LIN {X 0,Y 171.569,Z 534.537,A -85,B 0,C 180,E1 -24803.925,E2 -24803.925} C_VEL
LIN {X 0,Y 171.044,Z 531.437,A -85,B 0,C 180,E1 -24804.883,E2 -24804.883} C_VEL
LIN {X 0,Y 169.506,Z 526.594,A -85,B 0,C 180,E1 -24806.675,E2 -24806.675} C_VEL
LIN {X 0,Y 166.044,Z 528.715,A -85,B 0,C 180,E1 -24808.057,E2 -24808.057} C_VEL
LIN {X 0,Y 163.92,Z 529.698,A -85,B 0,C 180,E1 -24809.036,E2 -24809.036} C_VEL
LIN {X 0,Y 158.88,Z 534.272,A -85,B 0,C 180,E1 -24810.884,E2 -24810.884} C_VEL
LIN {X 0,Y 156.535,Z 535.959,A -85,B 0,C 180,E1 -24811.94,E2 -24811.94} C_VEL
LIN {X 0,Y 150.862,Z 538.736,A -85,B 0,C 180,E1 -24815.211,E2 -24815.211} C_VEL
LIN {X 0,Y 146.783,Z 541.804,A -85,B 0,C 180,E1 -24817.477,E2 -24817.477} C_VEL
LIN {X 0,Y 140.545,Z 545.035,A -85,B 0,C 180,E1 -24822.54,E2 -24822.54} C_VEL
LIN {X 0,Y 139.213,Z 546.109,A -85,B 0,C 180,E1 -24823.576,E2 -24823.576} C_VEL
LIN {X 0,Y 137.537,Z 547.231,A -85,B 0,C 180,E1 -24825.197,E2 -24825.197} C_VEL
LIN {X 0,Y 135.805,Z 547.355,A -85,B 0,C 180,E1 -24828.261,E2 -24828.261} C_VEL
LIN {X 0,Y 135.037,Z 555.759,A -85,B 0,C 180,E1 -24834.025,E2 -24834.025} C_VEL
LIN {X 0,Y 134.715,Z 562.924,A -85,B 0,C 180,E1 -24840,E2 -24840} C_VEL
LIN {X 0,Y 136.036,Z 570.119,A -85,B 0,C 180,E1 -24847.421,E2 -24847.421} C_VEL
LIN {X 0,Y 138.515,Z 574.658,A -85,B 0,C 180,E1 -24853.198,E2 -24853.198} C_VEL
LIN {X 0,Y 143.17,Z 578.949,A -85,B 0,C 180,E1 -24860.097,E2 -24860.097} C_VEL
LIN {X 0,Y 148.115,Z 581.35,A -85,B 0,C 180,E1 -24865.28,E2 -24865.28} C_VEL
LIN {X 0,Y 154.373,Z 582.922,A -85,B 0,C 180,E1 -24870.052,E2 -24870.052} C_VEL
LIN {X 0,Y 161.797,Z 583.682,A -85,B 0,C 180,E1 -24874.38,E2 -24874.38} C_VEL
LIN {X 0,Y 170.253,Z 583.595,A -85,B 0,C 180,E1 -24878.257,E2 -24878.257} C_VEL
LIN {X 0,Y 179.651,Z 582.767,A -85,B 0,C 180,E1 -24881.686,E2 -24881.686} C_VEL
LIN {X 0,Y 179.681,Z 582.884,A -85,B 0,C 180,E1 -24881.999,E2 -24881.999} C_VEL
LIN {X 0,Y 165.118,Z 588.068,A -85,B 0,C 180,E1 -24887.077,E2 -24887.077} C_VEL
LIN {X 0,Y 158.02,Z 590.446,A -85,B 0,C 180,E1 -24890.361,E2 -24890.361} C_VEL
LIN {X 0,Y 152.368,Z 599.787,A -85,B 0,C 180,E1 -24893.978,E2 -24893.978} C_VEL
LIN {X 0,Y 146.919,Z 608.149,A -85,B 0,C 180,E1 -24898.251,E2 -24898.251} C_VEL
LIN {X 0,Y 142.926,Z 614.092,A -85,B 0,C 180,E1 -24902.264,E2 -24902.264} C_VEL
LIN {X 0,Y 139.782,Z 618.749,A -85,B 0,C 180,E1 -24906.283,E2 -24906.283} C_VEL
LIN {X 0,Y 136.398,Z 623.68,A -85,B 0,C 180,E1 -24911.992,E2 -24911.992} C_VEL
LIN {X 0,Y 134.421,Z 627.109,A -85,B 0,C 180,E1 -24917.928,E2 -24917.928} C_VEL
LIN {X 0,Y 133.541,Z 629.139,A -85,B 0,C 180,E1 -24923.958,E2 -24923.958} C_VEL
LIN {X 0,Y 133.456,Z 629.808,A -85,B 0,C 180,E1 -24930,E2 -24930} C_VEL
LIN {X 0,Y 133.541,Z 629.118,A -85,B 0,C 180,E1 -24936.042,E2 -24936.042} C_VEL
LIN {X 0,Y 134.414,Z 627.073,A -85,B 0,C 180,E1 -24942.072,E2 -24942.072} C_VEL
LIN {X 0,Y 136.386,Z 623.622,A -85,B 0,C 180,E1 -24948.01,E2 -24948.01} C_VEL
LIN {X 0,Y 139.73,Z 618.666,A -85,B 0,C 180,E1 -24953.727,E2 -24953.727} C_VEL
LIN {X 0,Y 144.19,Z 612.057,A -85,B 0,C 180,E1 -24959.171,E2 -24959.171} C_VEL
LIN {X 0,Y 149.133,Z 604.663,A -85,B 0,C 180,E1 -24963.623,E2 -24963.623} C_VEL
LIN {X 0,Y 153.97,Z 596.923,A -85,B 0,C 180,E1 -24967.214,E2 -24967.214} C_VEL
LIN {X 0,Y 155.689,Z 594.039,A -85,B 0,C 180,E1 -24968.331,E2 -24968.331} C_VEL
LIN {X 0,Y 157.521,Z 590.227,A -85,B 0,C 180,E1 -24969.845,E2 -24969.845} C_VEL
LIN {X 0,Y 159.212,Z 583.792,A -85,B 0,C 180,E1 -24972.497,E2 -24972.497} C_VEL
LIN {X 0,Y 160.162,Z 578.388,A -85,B 0,C 180,E1 -24974.587,E2 -24974.587} C_VEL
LIN {X 0,Y 161.493,Z 572.56,A -85,B 0,C 180,E1 -24976.473,E2 -24976.473} C_VEL
LIN {X 0,Y 164.734,Z 560.752,A -85,B 0,C 180,E1 -24979.58,E2 -24979.58} C_VEL
LIN {X 0,Y 165.802,Z 555.433,A -85,B 0,C 180,E1 -24980.889,E2 -24980.889} C_VEL
LIN {X 0,Y 166.494,Z 546.263,A -85,B 0,C 180,E1 -24983.324,E2 -24983.324} C_VEL
LIN {X 0,Y 166.301,Z 536.113,A -85,B 0,C 180,E1 -24986.1,E2 -24986.1} C_VEL
LIN {X 0,Y 165.282,Z 526.155,A -85,B 0,C 180,E1 -24988.984,E2 -24988.984} C_VEL
LIN {X 0,Y 164.384,Z 521.991,A -85,B 0,C 180,E1 -24990.374,E2 -24990.374} C_VEL
LIN {X 0,Y 161.323,Z 513.981,A -85,B 0,C 180,E1 -24994,E2 -24994} C_VEL
LIN {X 0,Y 158.783,Z 508.688,A -85,B 0,C 180,E1 -24996.957,E2 -24996.957} C_VEL
LIN {X 0,Y 155.021,Z 503.691,A -85,B 0,C 180,E1 -25001.497,E2 -25001.497} C_VEL
LIN {X 0,Y 150.507,Z 497.984,A -85,B 0,C 180,E1 -25009.235,E2 -25009.235} C_VEL
LIN {X 0,Y 148.46,Z 496.298,A -85,B 0,C 180,E1 -25015.928,E2 -25015.928} C_VEL
LIN {X 0,Y 148.135,Z 496.053,A -85,B 0,C 180,E1 -25020.68,E2 -25020.68} C_VEL
LIN {X 0,Y 149.359,Z 498.244,A -85,B 0,C 180,E1 -25028.115,E2 -25028.115} C_VEL
LIN {X 0,Y 153.191,Z 504.707,A -85,B 0,C 180,E1 -25036.488,E2 -25036.488} C_VEL
LIN {X 0,Y 156.055,Z 509.696,A -85,B 0,C 180,E1 -25040.773,E2 -25040.773} C_VEL
LIN {X 0,Y 156.965,Z 511.228,A -85,B 0,C 180,E1 -25041.937,E2 -25041.937} C_VEL
LIN {X 0,Y 159.573,Z 516.438,A -85,B 0,C 180,E1 -25045.256,E2 -25045.256} C_VEL
LIN {X 0,Y 161.808,Z 521.62,A -85,B 0,C 180,E1 -25048.011,E2 -25048.011} C_VEL
LIN {X 0,Y 164.559,Z 529.199,A -85,B 0,C 180,E1 -25051.473,E2 -25051.473} C_VEL
LIN {X 0,Y 166.521,Z 536.003,A -85,B 0,C 180,E1 -25054.213,E2 -25054.213} C_VEL
LIN {X 0,Y 166.802,Z 539.563,A -85,B 0,C 180,E1 -25055.294,E2 -25055.294} C_VEL
LIN {X 0,Y 166.505,Z 549.955,A -85,B 0,C 180,E1 -25058.119,E2 -25058.119} C_VEL
LIN {X 0,Y 165.563,Z 558.499,A -85,B 0,C 180,E1 -25060.486,E2 -25060.486} C_VEL
LIN {X 0,Y 163.711,Z 568.454,A -85,B 0,C 180,E1 -25063.383,E2 -25063.383} C_VEL
LIN {X 0,Y 160.764,Z 574.861,A -85,B 0,C 180,E1 -25064.912,E2 -25064.912} C_VEL
LIN {X 0,Y 154.657,Z 585.764,A -85,B 0,C 180,E1 -25067.911,E2 -25067.911} C_VEL
LIN {X 0,Y 148.966,Z 595.031,A -85,B 0,C 180,E1 -25071.309,E2 -25071.309} C_VEL
LIN {X 0,Y 142.945,Z 603.841,A -85,B 0,C 180,E1 -25075.569,E2 -25075.569} C_VEL
LIN {X 0,Y 137.757,Z 610.923,A -85,B 0,C 180,E1 -25080.147,E2 -25080.147} C_VEL
LIN {X 0,Y 133.776,Z 616.611,A -85,B 0,C 180,E1 -25085.147,E2 -25085.147} C_VEL
LIN {X 0,Y 129.981,Z 621.53,A -85,B 0,C 180,E1 -25091.07,E2 -25091.07} C_VEL
LIN {X 0,Y 127.674,Z 624.95,A -85,B 0,C 180,E1 -25097.28,E2 -25097.28} C_VEL
LIN {X 0,Y 126.489,Z 626.977,A -85,B 0,C 180,E1 -25103.62,E2 -25103.62} C_VEL
LIN {X 0,Y 126.36,Z 627.665,A -85,B 0,C 180,E1 -25110,E2 -25110} C_VEL
LIN {X 0,Y 126.489,Z 627.022,A -85,B 0,C 180,E1 -25116.38,E2 -25116.38} C_VEL
LIN {X 0,Y 127.666,Z 625.03,A -85,B 0,C 180,E1 -25122.721,E2 -25122.721} C_VEL
LIN {X 0,Y 129.919,Z 621.65,A -85,B 0,C 180,E1 -25128.94,E2 -25128.94} C_VEL
LIN {X 0,Y 133.711,Z 616.777,A -85,B 0,C 180,E1 -25134.865,E2 -25134.865} C_VEL
LIN {X 0,Y 138.483,Z 610.261,A -85,B 0,C 180,E1 -25140.497,E2 -25140.497} C_VEL
LIN {X 0,Y 143.722,Z 602.985,A -85,B 0,C 180,E1 -25145.07,E2 -25145.07} C_VEL
LIN {X 0,Y 149.786,Z 593.909,A -85,B 0,C 180,E1 -25149.303,E2 -25149.303} C_VEL
LIN {X 0,Y 155.605,Z 584.409,A -85,B 0,C 180,E1 -25152.647,E2 -25152.647} C_VEL
LIN {X 0,Y 161.49,Z 573.747,A -85,B 0,C 180,E1 -25155.502,E2 -25155.502} C_VEL
LIN {X 0,Y 163.702,Z 568.999,A -85,B 0,C 180,E1 -25156.614,E2 -25156.614} C_VEL
LIN {X 0,Y 165.743,Z 558.201,A -85,B 0,C 180,E1 -25159.752,E2 -25159.752} C_VEL
LIN {X 0,Y 166.8,Z 547.36,A -85,B 0,C 180,E1 -25162.742,E2 -25162.742} C_VEL
LIN {X 0,Y 166.895,Z 537.118,A -85,B 0,C 180,E1 -25165.558,E2 -25165.558} C_VEL
LIN {X 0,Y 166.075,Z 534.53,A -85,B 0,C 180,E1 -25166.623,E2 -25166.623} C_VEL
LIN {X 0,Y 163.748,Z 535.647,A -85,B 0,C 180,E1 -25167.591,E2 -25167.591} C_VEL
LIN {X 0,Y 158.535,Z 539.947,A -85,B 0,C 180,E1 -25169.349,E2 -25169.349} C_VEL
LIN {X 0,Y 153.965,Z 542.753,A -85,B 0,C 180,E1 -25171.361,E2 -25171.361} C_VEL
LIN {X 0,Y 149.956,Z 544.53,A -85,B 0,C 180,E1 -25173.561,E2 -25173.561} C_VEL
LIN {X 0,Y 145.673,Z 547.346,A -85,B 0,C 180,E1 -25175.788,E2 -25175.788} C_VEL
LIN {X 0,Y 134.264,Z 553.473,A -85,B 0,C 180,E1 -25184.827,E2 -25184.827} C_VEL
LIN {X 0,Y 132.3,Z 554.047,A -85,B 0,C 180,E1 -25187.732,E2 -25187.732} C_VEL
LIN {X 0,Y 129.711,Z 556.293,A -85,B 0,C 180,E1 -25190.645,E2 -25190.645} C_VEL
LIN {X 0,Y 128.153,Z 557.299,A -85,B 0,C 180,E1 -25193.703,E2 -25193.703} C_VEL
LIN {X 0,Y 127.832,Z 557.367,A -85,B 0,C 180,E1 -25195.862,E2 -25195.862} C_VEL
LIN {X 0,Y 127.943,Z 565.324,A -85,B 0,C 180,E1 -25203.149,E2 -25203.149} C_VEL
LIN {X 0,Y 129.574,Z 570.963,A -85,B 0,C 180,E1 -25209.364,E2 -25209.364} C_VEL
LIN {X 0,Y 132.485,Z 575.527,A -85,B 0,C 180,E1 -25215.381,E2 -25215.381} C_VEL
LIN {X 0,Y 136.532,Z 579.09,A -85,B 0,C 180,E1 -25221.12,E2 -25221.12} C_VEL
LIN {X 0,Y 141.755,Z 581.845,A -85,B 0,C 180,E1 -25226.5,E2 -25226.5} C_VEL
LIN {X 0,Y 148.331,Z 583.708,A -85,B 0,C 180,E1 -25231.412,E2 -25231.412} C_VEL
LIN {X 0,Y 160.314,Z 585.061,A -85,B 0,C 180,E1 -25237.861,E2 -25237.861} C_VEL
LIN {X 0,Y 169.604,Z 584.916,A -85,B 0,C 180,E1 -25241.529,E2 -25241.529} C_VEL
LIN {X 0,Y 169.802,Z 585.004,A -85,B 0,C 180,E1 -25241.84,E2 -25241.84} C_VEL
LIN {X 0,Y 159.996,Z 587.947,A -85,B 0,C 180,E1 -25245.347,E2 -25245.347} C_VEL
LIN {X 0,Y 152.894,Z 589.992,A -85,B 0,C 180,E1 -25248.532,E2 -25248.532} C_VEL
LIN {X 0,Y 147.511,Z 598.388,A -85,B 0,C 180,E1 -25251.73,E2 -25251.73} C_VEL
LIN {X 0,Y 141.697,Z 606.984,A -85,B 0,C 180,E1 -25256.083,E2 -25256.083} C_VEL
LIN {X 0,Y 136.338,Z 614.467,A -85,B 0,C 180,E1 -25261.201,E2 -25261.201} C_VEL
LIN {X 0,Y 132.292,Z 620.108,A -85,B 0,C 180,E1 -25266.52,E2 -25266.52} C_VEL
LIN {X 0,Y 129.628,Z 623.622,A -85,B 0,C 180,E1 -25271.016,E2 -25271.016} C_VEL
LIN {X 0,Y 127.447,Z 627.051,A -85,B 0,C 180,E1 -25277.257,E2 -25277.257} C_VEL
LIN {X 0,Y 126.462,Z 629.081,A -85,B 0,C 180,E1 -25283.619,E2 -25283.619} C_VEL
LIN {X 0,Y 126.362,Z 629.75,A -85,B 0,C 180,E1 -25290,E2 -25290} C_VEL
LIN {X 0,Y 126.461,Z 629.059,A -85,B 0,C 180,E1 -25296.382,E2 -25296.382} C_VEL
LIN {X 0,Y 127.44,Z 627.013,A -85,B 0,C 180,E1 -25302.744,E2 -25302.744} C_VEL
LIN {X 0,Y 129.616,Z 623.563,A -85,B 0,C 180,E1 -25308.986,E2 -25308.986} C_VEL
LIN {X 0,Y 133.222,Z 618.607,A -85,B 0,C 180,E1 -25314.963,E2 -25314.963} C_VEL
LIN {X 0,Y 136.682,Z 613.761,A -85,B 0,C 180,E1 -25319.277,E2 -25319.277} C_VEL
LIN {X 0,Y 141.639,Z 606.852,A -85,B 0,C 180,E1 -25323.933,E2 -25323.933} C_VEL
LIN {X 0,Y 147.443,Z 598.225,A -85,B 0,C 180,E1 -25328.291,E2 -25328.291} C_VEL
LIN {X 0,Y 153.167,Z 589.19,A -85,B 0,C 180,E1 -25331.707,E2 -25331.707} C_VEL
LIN {X 0,Y 158.257,Z 580.174,A -85,B 0,C 180,E1 -25334.382,E2 -25334.382} C_VEL
LIN {X 0,Y 160.827,Z 574.699,A -85,B 0,C 180,E1 -25335.835,E2 -25335.835} C_VEL
LIN {X 0,Y 161.493,Z 572.56,A -85,B 0,C 180,E1 -25336.473,E2 -25336.473} C_VEL
LIN {X 0,Y 162.309,Z 568.2,A -85,B 0,C 180,E1 -25337.87,E2 -25337.87} C_VEL
LIN {X 0,Y 162.099,Z 561.494,A -85,B 0,C 180,E1 -25340.46,E2 -25340.46} C_VEL
LIN {X 0,Y 161.446,Z 553.277,A -85,B 0,C 180,E1 -25343.585,E2 -25343.585} C_VEL
LIN {X 0,Y 161.531,Z 550.221,A -85,B 0,C 180,E1 -25344.508,E2 -25344.508} C_VEL
LIN {X 0,Y 161.798,Z 539.321,A -85,B 0,C 180,E1 -25347.662,E2 -25347.662} C_VEL
LIN {X 0,Y 161.078,Z 529.294,A -85,B 0,C 180,E1 -25350.765,E2 -25350.765} C_VEL
LIN {X 0,Y 160.898,Z 527.698,A -85,B 0,C 180,E1 -25351.284,E2 -25351.284} C_VEL
LIN {X 0,Y 158.372,Z 519.868,A -85,B 0,C 180,E1 -25354.978,E2 -25354.978} C_VEL
LIN {X 0,Y 156.273,Z 514.897,A -85,B 0,C 180,E1 -25357.874,E2 -25357.874} C_VEL
LIN {X 0,Y 153.065,Z 510.194,A -85,B 0,C 180,E1 -25362.291,E2 -25362.291} C_VEL
LIN {X 0,Y 149.242,Z 504.86,A -85,B 0,C 180,E1 -25369.701,E2 -25369.701} C_VEL
LIN {X 0,Y 147.287,Z 503.093,A -85,B 0,C 180,E1 -25377.265,E2 -25377.265} C_VEL
LIN {X 0,Y 147.133,Z 503.104,A -85,B 0,C 180,E1 -25380.684,E2 -25380.684} C_VEL
LIN {X 0,Y 148.132,Z 505.12,A -85,B 0,C 180,E1 -25387.641,E2 -25387.641} C_VEL
LIN {X 0,Y 151.267,Z 511.307,A -85,B 0,C 180,E1 -25395.754,E2 -25395.754} C_VEL
LIN {X 0,Y 153.842,Z 516.272,A -85,B 0,C 180,E1 -25400.211,E2 -25400.211} C_VEL
LIN {X 0,Y 156.518,Z 522.246,A -85,B 0,C 180,E1 -25404.276,E2 -25404.276} C_VEL
LIN {X 0,Y 158.853,Z 528.646,A -85,B 0,C 180,E1 -25407.768,E2 -25407.768} C_VEL
LIN {X 0,Y 161.238,Z 536.757,A -85,B 0,C 180,E1 -25411.538,E2 -25411.538} C_VEL
LIN {X 0,Y 162.143,Z 541.835,A -85,B 0,C 180,E1 -25413.549,E2 -25413.549} C_VEL
LIN {X 0,Y 161.507,Z 551.754,A -85,B 0,C 180,E1 -25416.397,E2 -25416.397} C_VEL
LIN {X 0,Y 160.445,Z 559.918,A -85,B 0,C 180,E1 -25418.789,E2 -25418.789} C_VEL
LIN {X 0,Y 158.344,Z 569.601,A -85,B 0,C 180,E1 -25421.742,E2 -25421.742} C_VEL
LIN {X 0,Y 157.43,Z 571.865,A -85,B 0,C 180,E1 -25422.324,E2 -25422.324} C_VEL
LIN {X 0,Y 151.629,Z 582.302,A -85,B 0,C 180,E1 -25425.022,E2 -25425.022} C_VEL
LIN {X 0,Y 145.392,Z 592.16,A -85,B 0,C 180,E1 -25428.344,E2 -25428.344} C_VEL
LIN {X 0,Y 138.887,Z 601.554,A -85,B 0,C 180,E1 -25432.611,E2 -25432.611} C_VEL
LIN {X 0,Y 133.855,Z 608.144,A -85,B 0,C 180,E1 -25436.544,E2 -25436.544} C_VEL
LIN {X 0,Y 129.669,Z 613.608,A -85,B 0,C 180,E1 -25440.804,E2 -25440.804} C_VEL
LIN {X 0,Y 126.191,Z 618.078,A -85,B 0,C 180,E1 -25445.311,E2 -25445.311} C_VEL
LIN {X 0,Y 123.255,Z 621.589,A -85,B 0,C 180,E1 -25449.994,E2 -25449.994} C_VEL
LIN {X 0,Y 120.743,Z 625.009,A -85,B 0,C 180,E1 -25456.537,E2 -25456.537} C_VEL
LIN {X 0,Y 119.438,Z 627.036,A -85,B 0,C 180,E1 -25463.241,E2 -25463.241} C_VEL
LIN {X 0,Y 119.279,Z 627.724,A -85,B 0,C 180,E1 -25470,E2 -25470} C_VEL
LIN {X 0,Y 119.438,Z 627.08,A -85,B 0,C 180,E1 -25476.759,E2 -25476.759} C_VEL
LIN {X 0,Y 120.735,Z 625.088,A -85,B 0,C 180,E1 -25483.464,E2 -25483.464} C_VEL
LIN {X 0,Y 123.189,Z 621.708,A -85,B 0,C 180,E1 -25490.017,E2 -25490.017} C_VEL
LIN {X 0,Y 127.254,Z 616.834,A -85,B 0,C 180,E1 -25496.22,E2 -25496.22} C_VEL
LIN {X 0,Y 132.384,Z 610.316,A -85,B 0,C 180,E1 -25502.065,E2 -25502.065} C_VEL
LIN {X 0,Y 137.958,Z 603.038,A -85,B 0,C 180,E1 -25506.768,E2 -25506.768} C_VEL
LIN {X 0,Y 144.327,Z 593.961,A -85,B 0,C 180,E1 -25511.101,E2 -25511.101} C_VEL
LIN {X 0,Y 150.457,Z 584.457,A -85,B 0,C 180,E1 -25514.481,E2 -25514.481} C_VEL
LIN {X 0,Y 156.371,Z 574.21,A -85,B 0,C 180,E1 -25517.256,E2 -25517.256} C_VEL
LIN {X 0,Y 158.288,Z 570.221,A -85,B 0,C 180,E1 -25518.24,E2 -25518.24} C_VEL
LIN {X 0,Y 160.484,Z 560.426,A -85,B 0,C 180,E1 -25521.233,E2 -25521.233} C_VEL
LIN {X 0,Y 161.968,Z 548.715,A -85,B 0,C 180,E1 -25524.639,E2 -25524.639} C_VEL
LIN {X 0,Y 162.254,Z 542.389,A -85,B 0,C 180,E1 -25526.477,E2 -25526.477} C_VEL
LIN {X 0,Y 157.466,Z 545.916,A -85,B 0,C 180,E1 -25527.995,E2 -25527.995} C_VEL
LIN {X 0,Y 153.244,Z 548.341,A -85,B 0,C 180,E1 -25529.703,E2 -25529.703} C_VEL
LIN {X 0,Y 148.954,Z 550.207,A -85,B 0,C 180,E1 -25531.847,E2 -25531.847} C_VEL
LIN {X 0,Y 142.403,Z 553.912,A -85,B 0,C 180,E1 -25535.197,E2 -25535.197} C_VEL
LIN {X 0,Y 132.806,Z 558.559,A -85,B 0,C 180,E1 -25542.278,E2 -25542.278} C_VEL
LIN {X 0,Y 128.398,Z 560.578,A -85,B 0,C 180,E1 -25547.353,E2 -25547.353} C_VEL
LIN {X 0,Y 125.902,Z 562.354,A -85,B 0,C 180,E1 -25550.359,E2 -25550.359} C_VEL
LIN {X 0,Y 122.978,Z 564.389,A -85,B 0,C 180,E1 -25556.724,E2 -25556.724} C_VEL
LIN {X 0,Y 121.602,Z 566.135,A -85,B 0,C 180,E1 -25560,E2 -25560} C_VEL
LIN {X 0,Y 121.081,Z 567.203,A -85,B 0,C 180,E1 -25563.327,E2 -25563.327} C_VEL
LIN {X 0,Y 121.533,Z 567.585,A -85,B 0,C 180,E1 -25566.641,E2 -25566.641} C_VEL
LIN {X 0,Y 123.958,Z 572.967,A -85,B 0,C 180,E1 -25573.108,E2 -25573.108} C_VEL
LIN {X 0,Y 127.676,Z 577.34,A -85,B 0,C 180,E1 -25579.285,E2 -25579.285} C_VEL
LIN {X 0,Y 132.531,Z 580.754,A -85,B 0,C 180,E1 -25585.102,E2 -25585.102} C_VEL
LIN {X 0,Y 138.731,Z 583.367,A -85,B 0,C 180,E1 -25590.437,E2 -25590.437} C_VEL
LIN {X 0,Y 146.282,Z 585.18,A -85,B 0,C 180,E1 -25595.207,E2 -25595.207} C_VEL
LIN {X 0,Y 154.844,Z 586.184,A -85,B 0,C 180,E1 -25599.451,E2 -25599.451} C_VEL
LIN {X 0,Y 159.58,Z 586.409,A -85,B 0,C 180,E1 -25601.346,E2 -25601.346} C_VEL
LIN {X 0,Y 159.978,Z 586.483,A -85,B 0,C 180,E1 -25601.684,E2 -25601.684} C_VEL
LIN {X 0,Y 148.076,Z 589.337,A -85,B 0,C 180,E1 -25606.512,E2 -25606.512} C_VEL
LIN {X 0,Y 142.928,Z 596.985,A -85,B 0,C 180,E1 -25609.343,E2 -25609.343} C_VEL
LIN {X 0,Y 137.512,Z 604.695,A -85,B 0,C 180,E1 -25613.093,E2 -25613.093} C_VEL
LIN {X 0,Y 131.943,Z 612.051,A -85,B 0,C 180,E1 -25617.815,E2 -25617.815} C_VEL
LIN {X 0,Y 128.053,Z 617.17,A -85,B 0,C 180,E1 -25622.192,E2 -25622.192} C_VEL
LIN {X 0,Y 124.751,Z 621.298,A -85,B 0,C 180,E1 -25626.774,E2 -25626.774} C_VEL
LIN {X 0,Y 121.52,Z 625.459,A -85,B 0,C 180,E1 -25633.192,E2 -25633.192} C_VEL
LIN {X 0,Y 119.784,Z 628.179,A -85,B 0,C 180,E1 -25639.862,E2 -25639.862} C_VEL
LIN {X 0,Y 119.224,Z 629.526,A -85,B 0,C 180,E1 -25646.621,E2 -25646.621} C_VEL
LIN {X 0,Y 119.279,Z 629.691,A -85,B 0,C 180,E1 -25650,E2 -25650} C_VEL
LIN {X 0,Y 119.389,Z 629,A -85,B 0,C 180,E1 -25656.761,E2 -25656.761} C_VEL
LIN {X 0,Y 120.497,Z 626.954,A -85,B 0,C 180,E1 -25663.492,E2 -25663.492} C_VEL
LIN {X 0,Y 122.896,Z 623.504,A -85,B 0,C 180,E1 -25670.067,E2 -25670.067} C_VEL
LIN {X 0,Y 126.785,Z 618.548,A -85,B 0,C 180,E1 -25676.325,E2 -25676.325} C_VEL
LIN {X 0,Y 130.324,Z 613.922,A -85,B 0,C 180,E1 -25680.638,E2 -25680.638} C_VEL
LIN {X 0,Y 135.786,Z 606.794,A -85,B 0,C 180,E1 -25685.611,E2 -25685.611} C_VEL
LIN {X 0,Y 141.906,Z 598.168,A -85,B 0,C 180,E1 -25690.079,E2 -25690.079} C_VEL
LIN {X 0,Y 147.932,Z 589.135,A -85,B 0,C 180,E1 -25693.541,E2 -25693.541} C_VEL
LIN {X 0,Y 153.233,Z 580.12,A -85,B 0,C 180,E1 -25696.251,E2 -25696.251} C_VEL
LIN {X 0,Y 155.061,Z 576.646,A -85,B 0,C 180,E1 -25697.167,E2 -25697.167} C_VEL
LIN {X 0,Y 158.772,Z 565.171,A -85,B 0,C 180,E1 -25700.461,E2 -25700.461} C_VEL
LIN {X 0,Y 160.709,Z 557.267,A -85,B 0,C 180,E1 -25702.528,E2 -25702.528} C_VEL
LIN {X 0,Y 161.531,Z 550.221,A -85,B 0,C 180,E1 -25704.508,E2 -25704.508} C_VEL
LIN {X 0,Y 161.441,Z 545.854,A -85,B 0,C 180,E1 -25705.923,E2 -25705.923} C_VEL
LIN {X 0,Y 160.643,Z 542.049,A -85,B 0,C 180,E1 -25707.523,E2 -25707.523} C_VEL
LIN {X 0,Y 156.615,Z 530.782,A -85,B 0,C 180,E1 -25713.397,E2 -25713.397} C_VEL
LIN {X 0,Y 154.779,Z 524.499,A -85,B 0,C 180,E1 -25716.679,E2 -25716.679} C_VEL
LIN {X 0,Y 153.507,Z 520.932,A -85,B 0,C 180,E1 -25718.867,E2 -25718.867} C_VEL
LIN {X 0,Y 151.064,Z 516.879,A -85,B 0,C 180,E1 -25722.747,E2 -25722.747} C_VEL
LIN {X 0,Y 147.593,Z 511.6,A -85,B 0,C 180,E1 -25730.406,E2 -25730.406} C_VEL
LIN {X 0,Y 146.005,Z 510.072,A -85,B 0,C 180,E1 -25737.241,E2 -25737.241} C_VEL
LIN {X 0,Y 145.841,Z 510.098,A -85,B 0,C 180,E1 -25740.691,E2 -25740.691} C_VEL
LIN {X 0,Y 146.605,Z 512.01,A -85,B 0,C 180,E1 -25747.229,E2 -25747.229} C_VEL
LIN {X 0,Y 149.123,Z 517.912,A -85,B 0,C 180,E1 -25755.111,E2 -25755.111} C_VEL
LIN {X 0,Y 151.564,Z 523.402,A -85,B 0,C 180,E1 -25760.086,E2 -25760.086} C_VEL
LIN {X 0,Y 153.494,Z 528.698,A -85,B 0,C 180,E1 -25763.689,E2 -25763.689} C_VEL
LIN {X 0,Y 155.243,Z 534.319,A -85,B 0,C 180,E1 -25766.918,E2 -25766.918} C_VEL
LIN {X 0,Y 157.171,Z 542.633,A -85,B 0,C 180,E1 -25770.948,E2 -25770.948} C_VEL
LIN {X 0,Y 157.47,Z 545.173,A -85,B 0,C 180,E1 -25772.007,E2 -25772.007} C_VEL
LIN {X 0,Y 156.952,Z 551.537,A -85,B 0,C 180,E1 -25773.978,E2 -25773.978} C_VEL
LIN {X 0,Y 155.429,Z 561.339,A -85,B 0,C 180,E1 -25776.984,E2 -25776.984} C_VEL
LIN {X 0,Y 152.722,Z 571.917,A -85,B 0,C 180,E1 -25780.347,E2 -25780.347} C_VEL
LIN {X 0,Y 146.684,Z 582.356,A -85,B 0,C 180,E1 -25783.058,E2 -25783.058} C_VEL
LIN {X 0,Y 140.149,Z 592.216,A -85,B 0,C 180,E1 -25786.408,E2 -25786.408} C_VEL
LIN {X 0,Y 133.31,Z 601.611,A -85,B 0,C 180,E1 -25790.755,E2 -25790.755} C_VEL
LIN {X 0,Y 127.961,Z 608.202,A -85,B 0,C 180,E1 -25794.782,E2 -25794.782} C_VEL
LIN {X 0,Y 123.477,Z 613.666,A -85,B 0,C 180,E1 -25799.186,E2 -25799.186} C_VEL
LIN {X 0,Y 119.753,Z 618.137,A -85,B 0,C 180,E1 -25803.886,E2 -25803.886} C_VEL
LIN {X 0,Y 116.577,Z 621.648,A -85,B 0,C 180,E1 -25808.794,E2 -25808.794} C_VEL
LIN {X 0,Y 113.814,Z 625.068,A -85,B 0,C 180,E1 -25815.7,E2 -25815.7} C_VEL
LIN {X 0,Y 112.373,Z 627.095,A -85,B 0,C 180,E1 -25822.814,E2 -25822.814} C_VEL
LIN {X 0,Y 112.199,Z 627.782,A -85,B 0,C 180,E1 -25830,E2 -25830} C_VEL
LIN {X 0,Y 112.372,Z 627.138,A -85,B 0,C 180,E1 -25837.186,E2 -25837.186} C_VEL
LIN {X 0,Y 113.804,Z 625.146,A -85,B 0,C 180,E1 -25844.301,E2 -25844.301} C_VEL
LIN {X 0,Y 116.51,Z 621.765,A -85,B 0,C 180,E1 -25851.219,E2 -25851.219} C_VEL
LIN {X 0,Y 120.879,Z 616.89,A -85,B 0,C 180,E1 -25857.718,E2 -25857.718} C_VEL
LIN {X 0,Y 126.401,Z 610.371,A -85,B 0,C 180,E1 -25863.78,E2 -25863.78} C_VEL
LIN {X 0,Y 132.31,Z 603.092,A -85,B 0,C 180,E1 -25868.619,E2 -25868.619} C_VEL
LIN {X 0,Y 139.039,Z 594.012,A -85,B 0,C 180,E1 -25873.03,E2 -25873.03} C_VEL
LIN {X 0,Y 145.473,Z 584.506,A -85,B 0,C 180,E1 -25876.442,E2 -25876.442} C_VEL
LIN {X 0,Y 152.025,Z 573.486,A -85,B 0,C 180,E1 -25879.429,E2 -25879.429} C_VEL
LIN {X 0,Y 153.012,Z 571.43,A -85,B 0,C 180,E1 -25879.981,E2 -25879.981} C_VEL
LIN {X 0,Y 155.461,Z 561.739,A -85,B 0,C 180,E1 -25883.066,E2 -25883.066} C_VEL
LIN {X 0,Y 157.121,Z 551.323,A -85,B 0,C 180,E1 -25886.259,E2 -25886.259} C_VEL
LIN {X 0,Y 150.141,Z 554.811,A -85,B 0,C 180,E1 -25889.009,E2 -25889.009} C_VEL
LIN {X 0,Y 145.581,Z 556.82,A -85,B 0,C 180,E1 -25891.134,E2 -25891.134} C_VEL
LIN {X 0,Y 140.979,Z 559.254,A -85,B 0,C 180,E1 -25893.342,E2 -25893.342} C_VEL
LIN {X 0,Y 129.746,Z 564.295,A -85,B 0,C 180,E1 -25901.034,E2 -25901.034} C_VEL
LIN {X 0,Y 124.329,Z 566.677,A -85,B 0,C 180,E1 -25906.932,E2 -25906.932} C_VEL
LIN {X 0,Y 121.821,Z 568.217,A -85,B 0,C 180,E1 -25910.033,E2 -25910.033} C_VEL
LIN {X 0,Y 120.157,Z 569.118,A -85,B 0,C 180,E1 -25913.282,E2 -25913.282} C_VEL
LIN {X 0,Y 117.285,Z 571.906,A -85,B 0,C 180,E1 -25920,E2 -25920} C_VEL
LIN {X 0,Y 116.772,Z 572.855,A -85,B 0,C 180,E1 -25923.45,E2 -25923.45} C_VEL
LIN {X 0,Y 116.976,Z 573.42,A -85,B 0,C 180,E1 -25926.901,E2 -25926.901} C_VEL
LIN {X 0,Y 116.901,Z 574.842,A -85,B 0,C 180,E1 -25930.39,E2 -25930.39} C_VEL
LIN {X 0,Y 117.582,Z 575.864,A -85,B 0,C 180,E1 -25933.832,E2 -25933.832} C_VEL
LIN {X 0,Y 121.022,Z 577.073,A -85,B 0,C 180,E1 -25940.391,E2 -25940.391} C_VEL
LIN {X 0,Y 126.141,Z 580.829,A -85,B 0,C 180,E1 -25946.469,E2 -25946.469} C_VEL
LIN {X 0,Y 132.679,Z 583.71,A -85,B 0,C 180,E1 -25951.985,E2 -25951.985} C_VEL
LIN {X 0,Y 144.917,Z 586.64,A -85,B 0,C 180,E1 -25959.084,E2 -25959.084} C_VEL
LIN {X 0,Y 150.238,Z 587.319,A -85,B 0,C 180,E1 -25961.542,E2 -25961.542} C_VEL
LIN {X 0,Y 143.443,Z 588.681,A -85,B 0,C 180,E1 -25964.355,E2 -25964.355} C_VEL
LIN {X 0,Y 137.604,Z 596.933,A -85,B 0,C 180,E1 -25967.411,E2 -25967.411} C_VEL
LIN {X 0,Y 131.872,Z 604.641,A -85,B 0,C 180,E1 -25971.229,E2 -25971.229} C_VEL
LIN {X 0,Y 125.949,Z 611.995,A -85,B 0,C 180,E1 -25976.082,E2 -25976.082} C_VEL
LIN {X 0,Y 121.778,Z 617.114,A -85,B 0,C 180,E1 -25980.623,E2 -25980.623} C_VEL
LIN {X 0,Y 118.235,Z 621.241,A -85,B 0,C 180,E1 -25985.412,E2 -25985.412} C_VEL
LIN {X 0,Y 114.692,Z 625.401,A -85,B 0,C 180,E1 -25992.158,E2 -25992.158} C_VEL
LIN {X 0,Y 112.774,Z 628.12,A -85,B 0,C 180,E1 -25999.225,E2 -25999.225} C_VEL
LIN {X 0,Y 112.133,Z 629.468,A -85,B 0,C 180,E1 -26006.407,E2 -26006.407} C_VEL
LIN {X 0,Y 112.198,Z 629.633,A -85,B 0,C 180,E1 -26010,E2 -26010} C_VEL
LIN {X 0,Y 112.313,Z 628.941,A -85,B 0,C 180,E1 -26017.189,E2 -26017.189} C_VEL
LIN {X 0,Y 113.583,Z 626.895,A -85,B 0,C 180,E1 -26024.33,E2 -26024.33} C_VEL
LIN {X 0,Y 116.231,Z 623.445,A -85,B 0,C 180,E1 -26031.272,E2 -26031.272} C_VEL
LIN {X 0,Y 120.429,Z 618.49,A -85,B 0,C 180,E1 -26037.831,E2 -26037.831} C_VEL
LIN {X 0,Y 124.376,Z 613.683,A -85,B 0,C 180,E1 -26042.467,E2 -26042.467} C_VEL
LIN {X 0,Y 130.059,Z 606.737,A -85,B 0,C 180,E1 -26047.439,E2 -26047.439} C_VEL
LIN {X 0,Y 136.523,Z 598.112,A -85,B 0,C 180,E1 -26052.007,E2 -26052.007} C_VEL
LIN {X 0,Y 142.861,Z 589.08,A -85,B 0,C 180,E1 -26055.506,E2 -26055.506} C_VEL
LIN {X 0,Y 148.867,Z 579.246,A -85,B 0,C 180,E1 -26058.466,E2 -26058.466} C_VEL
LIN {X 0,Y 150.258,Z 576.21,A -85,B 0,C 180,E1 -26059.366,E2 -26059.366} C_VEL
LIN {X 0,Y 154.322,Z 564.495,A -85,B 0,C 180,E1 -26062.77,E2 -26062.77} C_VEL
LIN {X 0,Y 155.752,Z 558.894,A -85,B 0,C 180,E1 -26064.313,E2 -26064.313} C_VEL
LIN {X 0,Y 156.982,Z 549.701,A -85,B 0,C 180,E1 -26067.067,E2 -26067.067} C_VEL
LIN {X 0,Y 157.325,Z 540.304,A -85,B 0,C 180,E1 -26069.997,E2 -26069.997} C_VEL
LIN {X 0,Y 157.012,Z 532.27,A -85,B 0,C 180,E1 -26072.69,E2 -26072.69} C_VEL
LIN {X 0,Y 156.615,Z 530.782,A -85,B 0,C 180,E1 -26073.397,E2 -26073.397} C_VEL
LIN {X 0,Y 155.321,Z 527.894,A -85,B 0,C 180,E1 -26075.224,E2 -26075.224} C_VEL
LIN {X 0,Y 153.606,Z 526.098,A -85,B 0,C 180,E1 -26077.231,E2 -26077.231} C_VEL
LIN {X 0,Y 148.023,Z 522.596,A -85,B 0,C 180,E1 -26084.551,E2 -26084.551} C_VEL
LIN {X 0,Y 145.695,Z 518.338,A -85,B 0,C 180,E1 -26090.981,E2 -26090.981} C_VEL
LIN {X 0,Y 144.388,Z 517.006,A -85,B 0,C 180,E1 -26097.21,E2 -26097.21} C_VEL
LIN {X 0,Y 144.219,Z 517.022,A -85,B 0,C 180,E1 -26100.698,E2 -26100.698} C_VEL
LIN {X 0,Y 144.76,Z 518.811,A -85,B 0,C 180,E1 -26106.796,E2 -26106.796} C_VEL
LIN {X 0,Y 146.535,Z 523.752,A -85,B 0,C 180,E1 -26113.875,E2 -26113.875} C_VEL
LIN {X 0,Y 148.406,Z 528.759,A -85,B 0,C 180,E1 -26118.713,E2 -26118.713} C_VEL
LIN {X 0,Y 150.061,Z 534.321,A -85,B 0,C 180,E1 -26122.69,E2 -26122.69} C_VEL
LIN {X 0,Y 151.236,Z 538.835,A -85,B 0,C 180,E1 -26125.458,E2 -26125.458} C_VEL
LIN {X 0,Y 152.432,Z 545.234,A -85,B 0,C 180,E1 -26128.835,E2 -26128.835} C_VEL
LIN {X 0,Y 152.85,Z 549.462,A -85,B 0,C 180,E1 -26130.751,E2 -26130.751} C_VEL
LIN {X 0,Y 151.323,Z 559.099,A -85,B 0,C 180,E1 -26133.871,E2 -26133.871} C_VEL
LIN {X 0,Y 149.143,Z 567.97,A -85,B 0,C 180,E1 -26136.766,E2 -26136.766} C_VEL
LIN {X 0,Y 147.589,Z 573.018,A -85,B 0,C 180,E1 -26138.49,E2 -26138.49} C_VEL
LIN {X 0,Y 141.928,Z 582.41,A -85,B 0,C 180,E1 -26140.961,E2 -26140.961} C_VEL
LIN {X 0,Y 135.082,Z 592.272,A -85,B 0,C 180,E1 -26144.325,E2 -26144.325} C_VEL
LIN {X 0,Y 127.88,Z 601.668,A -85,B 0,C 180,E1 -26148.739,E2 -26148.739} C_VEL
LIN {X 0,Y 122.217,Z 608.26,A -85,B 0,C 180,E1 -26152.858,E2 -26152.858} C_VEL
LIN {X 0,Y 117.394,Z 613.725,A -85,B 0,C 180,E1 -26157.398,E2 -26157.398} C_VEL
LIN {X 0,Y 112.164,Z 619.442,A -85,B 0,C 180,E1 -26163.985,E2 -26163.985} C_VEL
LIN {X 0,Y 108.266,Z 623.597,A -85,B 0,C 180,E1 -26171.06,E2 -26171.06} C_VEL
LIN {X 0,Y 105.973,Z 626.31,A -85,B 0,C 180,E1 -26178.524,E2 -26178.524} C_VEL
LIN {X 0,Y 105.048,Z 627.664,A -85,B 0,C 180,E1 -26186.164,E2 -26186.164} C_VEL
LIN {X 0,Y 105.106,Z 627.84,A -85,B 0,C 180,E1 -26190,E2 -26190} C_VEL
LIN {X 0,Y 105.317,Z 627.196,A -85,B 0,C 180,E1 -26197.67,E2 -26197.67} C_VEL
LIN {X 0,Y 106.913,Z 625.203,A -85,B 0,C 180,E1 -26205.245,E2 -26205.245} C_VEL
LIN {X 0,Y 109.892,Z 621.822,A -85,B 0,C 180,E1 -26212.564,E2 -26212.564} C_VEL
LIN {X 0,Y 114.598,Z 616.947,A -85,B 0,C 180,E1 -26219.381,E2 -26219.381} C_VEL
LIN {X 0,Y 120.542,Z 610.427,A -85,B 0,C 180,E1 -26225.664,E2 -26225.664} C_VEL
LIN {X 0,Y 126.826,Z 603.145,A -85,B 0,C 180,E1 -26230.626,E2 -26230.626} C_VEL
LIN {X 0,Y 132.86,Z 595.506,A -85,B 0,C 180,E1 -26234.499,E2 -26234.499} C_VEL
LIN {X 0,Y 139.518,Z 586.308,A -85,B 0,C 180,E1 -26237.988,E2 -26237.988} C_VEL
LIN {X 0,Y 146.169,Z 575.867,A -85,B 0,C 180,E1 -26240.961,E2 -26240.961} C_VEL
LIN {X 0,Y 148.121,Z 571.945,A -85,B 0,C 180,E1 -26242.051,E2 -26242.051} C_VEL
LIN {X 0,Y 150.893,Z 561.783,A -85,B 0,C 180,E1 -26245.44,E2 -26245.44} C_VEL
LIN {X 0,Y 151.342,Z 559.662,A -85,B 0,C 180,E1 -26246.134,E2 -26246.134} C_VEL
LIN {X 0,Y 146.789,Z 561.08,A -85,B 0,C 180,E1 -26248.22,E2 -26248.22} C_VEL
LIN {X 0,Y 137.3,Z 565.391,A -85,B 0,C 180,E1 -26252.568,E2 -26252.568} C_VEL
LIN {X 0,Y 125.705,Z 570.15,A -85,B 0,C 180,E1 -26260.4,E2 -26260.4} C_VEL
LIN {X 0,Y 117.487,Z 573.857,A -85,B 0,C 180,E1 -26269.662,E2 -26269.662} C_VEL
LIN {X 0,Y 115.693,Z 574.797,A -85,B 0,C 180,E1 -26273.021,E2 -26273.021} C_VEL
LIN {X 0,Y 112.471,Z 577.746,A -85,B 0,C 180,E1 -26281.164,E2 -26281.164} C_VEL
LIN {X 0,Y 112.258,Z 579.005,A -85,B 0,C 180,E1 -26287.193,E2 -26287.193} C_VEL
LIN {X 0,Y 112.254,Z 580.28,A -85,B 0,C 180,E1 -26290.826,E2 -26290.826} C_VEL
LIN {X 0,Y 112.995,Z 581.221,A -85,B 0,C 180,E1 -26294.406,E2 -26294.406} C_VEL
LIN {X 0,Y 116.39,Z 582.369,A -85,B 0,C 180,E1 -26301.241,E2 -26301.241} C_VEL
LIN {X 0,Y 120.593,Z 584.305,A -85,B 0,C 180,E1 -26307.79,E2 -26307.79} C_VEL
LIN {X 0,Y 126.9,Z 585.428,A -85,B 0,C 180,E1 -26313.629,E2 -26313.629} C_VEL
LIN {X 0,Y 133.791,Z 586.049,A -85,B 0,C 180,E1 -26318.018,E2 -26318.018} C_VEL
LIN {X 0,Y 140.57,Z 587.476,A -85,B 0,C 180,E1 -26321.414,E2 -26321.414} C_VEL
LIN {X 0,Y 139.186,Z 587.81,A -85,B 0,C 180,E1 -26321.995,E2 -26321.995} C_VEL
LIN {X 0,Y 133.494,Z 595.42,A -85,B 0,C 180,E1 -26324.706,E2 -26324.706} C_VEL
LIN {X 0,Y 127.358,Z 603.367,A -85,B 0,C 180,E1 -26328.532,E2 -26328.532} C_VEL
LIN {X 0,Y 121.774,Z 609.971,A -85,B 0,C 180,E1 -26332.7,E2 -26332.7} C_VEL
LIN {X 0,Y 116.969,Z 615.45,A -85,B 0,C 180,E1 -26337.265,E2 -26337.265} C_VEL
LIN {X 0,Y 111.773,Z 621.184,A -85,B 0,C 180,E1 -26343.887,E2 -26343.887} C_VEL
LIN {X 0,Y 107.909,Z 625.343,A -85,B 0,C 180,E1 -26350.995,E2 -26350.995} C_VEL
LIN {X 0,Y 105.793,Z 628.062,A -85,B 0,C 180,E1 -26358.504,E2 -26358.504} C_VEL
LIN {X 0,Y 105.042,Z 629.41,A -85,B 0,C 180,E1 -26366.164,E2 -26366.164} C_VEL
LIN {X 0,Y 105.105,Z 629.574,A -85,B 0,C 180,E1 -26370,E2 -26370} C_VEL
LIN {X 0,Y 105.26,Z 628.882,A -85,B 0,C 180,E1 -26377.674,E2 -26377.674} C_VEL
LIN {X 0,Y 106.667,Z 626.836,A -85,B 0,C 180,E1 -26385.281,E2 -26385.281} C_VEL
LIN {X 0,Y 109.626,Z 623.386,A -85,B 0,C 180,E1 -26392.622,E2 -26392.622} C_VEL
LIN {X 0,Y 114.16,Z 618.431,A -85,B 0,C 180,E1 -26399.505,E2 -26399.505} C_VEL
LIN {X 0,Y 118.422,Z 613.625,A -85,B 0,C 180,E1 -26404.319,E2 -26404.319} C_VEL
LIN {X 0,Y 124.456,Z 606.679,A -85,B 0,C 180,E1 -26409.441,E2 -26409.441} C_VEL
LIN {X 0,Y 131.31,Z 598.055,A -85,B 0,C 180,E1 -26414.09,E2 -26414.09} C_VEL
LIN {X 0,Y 137.972,Z 589.024,A -85,B 0,C 180,E1 -26417.613,E2 -26417.613} C_VEL
LIN {X 0,Y 143.679,Z 580.104,A -85,B 0,C 180,E1 -26420.339,E2 -26420.339} C_VEL
LIN {X 0,Y 145.617,Z 575.941,A -85,B 0,C 180,E1 -26421.655,E2 -26421.655} C_VEL
LIN {X 0,Y 149.898,Z 564.522,A -85,B 0,C 180,E1 -26425.019,E2 -26425.019} C_VEL
LIN {X 0,Y 151.504,Z 557.664,A -85,B 0,C 180,E1 -26427.121,E2 -26427.121} C_VEL
LIN {X 0,Y 152.57,Z 550.092,A -85,B 0,C 180,E1 -26429.556,E2 -26429.556} C_VEL
LIN {X 0,Y 153.127,Z 540.696,A -85,B 0,C 180,E1 -26432.68,E2 -26432.68} C_VEL
LIN {X 0,Y 153.177,Z 538.157,A -85,B 0,C 180,E1 -26433.574,E2 -26433.574} C_VEL
LIN {X 0,Y 152.506,Z 534.104,A -85,B 0,C 180,E1 -26435.497,E2 -26435.497} C_VEL
LIN {X 0,Y 151.226,Z 529.197,A -85,B 0,C 180,E1 -26438.352,E2 -26438.352} C_VEL
LIN {X 0,Y 150.793,Z 527.483,A -85,B 0,C 180,E1 -26439.398,E2 -26439.398} C_VEL
LIN {X 0,Y 148.672,Z 523.415,A -85,B 0,C 180,E1 -26443.347,E2 -26443.347} C_VEL
LIN {X 0,Y 148.023,Z 522.596,A -85,B 0,C 180,E1 -26444.551,E2 -26444.551} C_VEL
LIN {X 0,Y 146.803,Z 521.78,A -85,B 0,C 180,E1 -26446.779,E2 -26446.779} C_VEL
LIN {X 0,Y 145.48,Z 522.023,A -85,B 0,C 180,E1 -26449.056,E2 -26449.056} C_VEL
LIN {X 0,Y 142.724,Z 523.947,A -85,B 0,C 180,E1 -26455.318,E2 -26455.318} C_VEL
LIN {X 0,Y 142.467,Z 523.883,A -85,B 0,C 180,E1 -26456.93,E2 -26456.93} C_VEL
LIN {X 0,Y 142.27,Z 523.862,A -85,B 0,C 180,E1 -26460.708,E2 -26460.708} C_VEL
LIN {X 0,Y 142.549,Z 525.155,A -85,B 0,C 180,E1 -26465.659,E2 -26465.659} C_VEL
LIN {X 0,Y 143.734,Z 529.832,A -85,B 0,C 180,E1 -26472.711,E2 -26472.711} C_VEL
LIN {X 0,Y 145.305,Z 534.865,A -85,B 0,C 180,E1 -26477.92,E2 -26477.92} C_VEL
LIN {X 0,Y 146.52,Z 540.068,A -85,B 0,C 180,E1 -26481.823,E2 -26481.823} C_VEL
LIN {X 0,Y 147.502,Z 545.298,A -85,B 0,C 180,E1 -26485.138,E2 -26485.138} C_VEL
LIN {X 0,Y 148.232,Z 552.022,A -85,B 0,C 180,E1 -26488.766,E2 -26488.766} C_VEL
LIN {X 0,Y 147.726,Z 555.935,A -85,B 0,C 180,E1 -26490.207,E2 -26490.207} C_VEL
LIN {X 0,Y 145.466,Z 565.47,A -85,B 0,C 180,E1 -26493.453,E2 -26493.453} C_VEL
LIN {X 0,Y 142.568,Z 574.233,A -85,B 0,C 180,E1 -26496.535,E2 -26496.535} C_VEL
LIN {X 0,Y 136.141,Z 584.223,A -85,B 0,C 180,E1 -26499.254,E2 -26499.254} C_VEL
LIN {X 0,Y 130.191,Z 592.328,A -85,B 0,C 180,E1 -26502.076,E2 -26502.076} C_VEL
LIN {X 0,Y 123.639,Z 600.508,A -85,B 0,C 180,E1 -26505.867,E2 -26505.867} C_VEL
LIN {X 0,Y 116.612,Z 608.318,A -85,B 0,C 180,E1 -26510.742,E2 -26510.742} C_VEL
LIN {X 0,Y 111.433,Z 613.784,A -85,B 0,C 180,E1 -26515.415,E2 -26515.415} C_VEL
LIN {X 0,Y 105.806,Z 619.501,A -85,B 0,C 180,E1 -26522.292,E2 -26522.292} C_VEL
LIN {X 0,Y 101.551,Z 623.656,A -85,B 0,C 180,E1 -26529.755,E2 -26529.755} C_VEL
LIN {X 0,Y 99.002,Z 626.369,A -85,B 0,C 180,E1 -26537.704,E2 -26537.704} C_VEL
LIN {X 0,Y 97.955,Z 627.723,A -85,B 0,C 180,E1 -26545.886,E2 -26545.886} C_VEL
LIN {X 0,Y 98.006,Z 627.899,A -85,B 0,C 180,E1 -26550,E2 -26550} C_VEL
LIN {X 0,Y 98.287,Z 627.254,A -85,B 0,C 180,E1 -26558.222,E2 -26558.222} C_VEL
LIN {X 0,Y 100.063,Z 625.261,A -85,B 0,C 180,E1 -26566.316,E2 -26566.316} C_VEL
LIN {X 0,Y 103.35,Z 621.879,A -85,B 0,C 180,E1 -26574.08,E2 -26574.08} C_VEL
LIN {X 0,Y 108.429,Z 617.003,A -85,B 0,C 180,E1 -26581.234,E2 -26581.234} C_VEL
LIN {X 0,Y 114.812,Z 610.482,A -85,B 0,C 180,E1 -26587.744,E2 -26587.744} C_VEL
LIN {X 0,Y 121.511,Z 603.199,A -85,B 0,C 180,E1 -26592.812,E2 -26592.812} C_VEL
LIN {X 0,Y 128.977,Z 594.115,A -85,B 0,C 180,E1 -26597.36,E2 -26597.36} C_VEL
LIN {X 0,Y 136.062,Z 584.603,A -85,B 0,C 180,E1 -26600.786,E2 -26600.786} C_VEL
LIN {X 0,Y 142.501,Z 574.613,A -85,B 0,C 180,E1 -26603.544,E2 -26603.544} C_VEL
LIN {X 0,Y 144.678,Z 568.518,A -85,B 0,C 180,E1 -26605.67,E2 -26605.67} C_VEL
LIN {X 0,Y 144.671,Z 566.651,A -85,B 0,C 180,E1 -26606.689,E2 -26606.689} C_VEL
LIN {X 0,Y 133.387,Z 571.319,A -85,B 0,C 180,E1 -26611.692,E2 -26611.692} C_VEL
LIN {X 0,Y 121.424,Z 575.784,A -85,B 0,C 180,E1 -26619.679,E2 -26619.679} C_VEL
LIN {X 0,Y 109.182,Z 581.523,A -85,B 0,C 180,E1 -26636.309,E2 -26636.309} C_VEL
LIN {X 0,Y 107.841,Z 582.76,A -85,B 0,C 180,E1 -26640,E2 -26640} C_VEL
LIN {X 0,Y 107.309,Z 584.318,A -85,B 0,C 180,E1 -26647.526,E2 -26647.526} C_VEL
LIN {X 0,Y 107.368,Z 585.478,A -85,B 0,C 180,E1 -26651.325,E2 -26651.325} C_VEL
LIN {X 0,Y 108.192,Z 586.331,A -85,B 0,C 180,E1 -26655.06,E2 -26655.06} C_VEL
LIN {X 0,Y 111.657,Z 587.51,A -85,B 0,C 180,E1 -26662.188,E2 -26662.188} C_VEL
LIN {X 0,Y 116.095,Z 589.284,A -85,B 0,C 180,E1 -26668.966,E2 -26668.966} C_VEL
LIN {X 0,Y 122.658,Z 590.343,A -85,B 0,C 180,E1 -26674.958,E2 -26674.958} C_VEL
LIN {X 0,Y 131.408,Z 591.022,A -85,B 0,C 180,E1 -26680.513,E2 -26680.513} C_VEL
LIN {X 0,Y 130.94,Z 592.409,A -85,B 0,C 180,E1 -26681.286,E2 -26681.286} C_VEL
LIN {X 0,Y 124.194,Z 600.859,A -85,B 0,C 180,E1 -26684.979,E2 -26684.979} C_VEL
LIN {X 0,Y 117.138,Z 608.914,A -85,B 0,C 180,E1 -26689.836,E2 -26689.836} C_VEL
LIN {X 0,Y 110.655,Z 615.771,A -85,B 0,C 180,E1 -26695.656,E2 -26695.656} C_VEL
LIN {X 0,Y 105.389,Z 621.127,A -85,B 0,C 180,E1 -26702.173,E2 -26702.173} C_VEL
LIN {X 0,Y 101.18,Z 625.286,A -85,B 0,C 180,E1 -26709.678,E2 -26709.678} C_VEL
LIN {X 0,Y 98.806,Z 628.004,A -85,B 0,C 180,E1 -26717.679,E2 -26717.679} C_VEL
LIN {X 0,Y 97.947,Z 629.351,A -85,B 0,C 180,E1 -26725.885,E2 -26725.885} C_VEL
LIN {X 0,Y 98.005,Z 629.516,A -85,B 0,C 180,E1 -26730,E2 -26730} C_VEL
LIN {X 0,Y 98.209,Z 628.823,A -85,B 0,C 180,E1 -26738.229,E2 -26738.229} C_VEL
LIN {X 0,Y 99.788,Z 626.777,A -85,B 0,C 180,E1 -26746.363,E2 -26746.363} C_VEL
LIN {X 0,Y 103.089,Z 623.327,A -85,B 0,C 180,E1 -26754.145,E2 -26754.145} C_VEL
LIN {X 0,Y 107.997,Z 618.372,A -85,B 0,C 180,E1 -26761.373,E2 -26761.373} C_VEL
LIN {X 0,Y 112.58,Z 613.566,A -85,B 0,C 180,E1 -26766.374,E2 -26766.374} C_VEL
LIN {X 0,Y 119.014,Z 606.621,A -85,B 0,C 180,E1 -26771.631,E2 -26771.631} C_VEL
LIN {X 0,Y 126.285,Z 597.998,A -85,B 0,C 180,E1 -26776.342,E2 -26776.342} C_VEL
LIN {X 0,Y 133.283,Z 588.97,A -85,B 0,C 180,E1 -26779.87,E2 -26779.87} C_VEL
LIN {X 0,Y 138.666,Z 580.949,A -85,B 0,C 180,E1 -26782.353,E2 -26782.353} C_VEL
LIN {X 0,Y 141.63,Z 574.824,A -85,B 0,C 180,E1 -26784.348,E2 -26784.348} C_VEL
LIN {X 0,Y 145.217,Z 565.922,A -85,B 0,C 180,E1 -26787.024,E2 -26787.024} C_VEL
LIN {X 0,Y 147.226,Z 558.012,A -85,B 0,C 180,E1 -26789.602,E2 -26789.602} C_VEL
LIN {X 0,Y 148.612,Z 548.889,A -85,B 0,C 180,E1 -26792.745,E2 -26792.745} C_VEL
LIN {X 0,Y 149.113,Z 542.913,A -85,B 0,C 180,E1 -26794.901,E2 -26794.901} C_VEL
LIN {X 0,Y 148.886,Z 539.904,A -85,B 0,C 180,E1 -26796.345,E2 -26796.345} C_VEL
LIN {X 0,Y 148.148,Z 535.749,A -85,B 0,C 180,E1 -26798.777,E2 -26798.777} C_VEL
LIN {X 0,Y 147.549,Z 533.19,A -85,B 0,C 180,E1 -26800.524,E2 -26800.524} C_VEL
LIN {X 0,Y 146.334,Z 530.393,A -85,B 0,C 180,E1 -26803.252,E2 -26803.252} C_VEL
LIN {X 0,Y 143.508,Z 524.978,A -85,B 0,C 180,E1 -26811.552,E2 -26811.552} C_VEL
LIN {X 0,Y 142.467,Z 523.883,A -85,B 0,C 180,E1 -26816.93,E2 -26816.93} C_VEL
LIN {X 0,Y 142.276,Z 524.01,A -85,B 0,C 180,E1 -26818.504,E2 -26818.504} C_VEL
LIN {X 0,Y 141.794,Z 525.428,A -85,B 0,C 180,E1 -26820.812,E2 -26820.812} C_VEL
LIN {X 0,Y 141.17,Z 527.738,A -85,B 0,C 180,E1 -26823.028,E2 -26823.028} C_VEL
LIN {X 0,Y 140.29,Z 532.954,A -85,B 0,C 180,E1 -26827.541,E2 -26827.541} C_VEL
LIN {X 0,Y 140.329,Z 534.228,A -85,B 0,C 180,E1 -26829.122,E2 -26829.122} C_VEL
LIN {X 0,Y 141.048,Z 536.943,A -85,B 0,C 180,E1 -26832.957,E2 -26832.957} C_VEL
LIN {X 0,Y 142.018,Z 541.036,A -85,B 0,C 180,E1 -26837.273,E2 -26837.273} C_VEL
LIN {X 0,Y 142.961,Z 546.625,A -85,B 0,C 180,E1 -26841.634,E2 -26841.634} C_VEL
LIN {X 0,Y 143.514,Z 552.897,A -85,B 0,C 180,E1 -26845.551,E2 -26845.551} C_VEL
LIN {X 0,Y 143.558,Z 556.914,A -85,B 0,C 180,E1 -26847.717,E2 -26847.717} C_VEL
LIN {X 0,Y 140.898,Z 566.832,A -85,B 0,C 180,E1 -26851.271,E2 -26851.271} C_VEL
LIN {X 0,Y 137.644,Z 575.61,A -85,B 0,C 180,E1 -26854.491,E2 -26854.491} C_VEL
LIN {X 0,Y 130.493,Z 586.037,A -85,B 0,C 180,E1 -26857.402,E2 -26857.402} C_VEL
LIN {X 0,Y 123.197,Z 595.314,A -85,B 0,C 180,E1 -26860.898,E2 -26860.898} C_VEL
LIN {X 0,Y 115.357,Z 604.128,A -85,B 0,C 180,E1 -26865.523,E2 -26865.523} C_VEL
LIN {X 0,Y 109.242,Z 610.345,A -85,B 0,C 180,E1 -26869.958,E2 -26869.958} C_VEL
LIN {X 0,Y 103.993,Z 615.437,A -85,B 0,C 180,E1 -26874.939,E2 -26874.939} C_VEL
LIN {X 0,Y 99.555,Z 619.56,A -85,B 0,C 180,E1 -26880.386,E2 -26880.386} C_VEL
LIN {X 0,Y 94.879,Z 623.715,A -85,B 0,C 180,E1 -26888.262,E2 -26888.262} C_VEL
LIN {X 0,Y 92.066,Z 626.428,A -85,B 0,C 180,E1 -26896.761,E2 -26896.761} C_VEL
LIN {X 0,Y 90.886,Z 627.781,A -85,B 0,C 180,E1 -26905.565,E2 -26905.565} C_VEL
LIN {X 0,Y 90.914,Z 627.957,A -85,B 0,C 180,E1 -26910,E2 -26910} C_VEL
LIN {X 0,Y 91.256,Z 627.313,A -85,B 0,C 180,E1 -26918.86,E2 -26918.86} C_VEL
LIN {X 0,Y 93.242,Z 625.319,A -85,B 0,C 180,E1 -26927.547,E2 -26927.547} C_VEL
LIN {X 0,Y 96.896,Z 621.937,A -85,B 0,C 180,E1 -26935.797,E2 -26935.797} C_VEL
LIN {X 0,Y 102.394,Z 617.06,A -85,B 0,C 180,E1 -26943.305,E2 -26943.305} C_VEL
LIN {X 0,Y 107.293,Z 612.448,A -85,B 0,C 180,E1 -26948.321,E2 -26948.321} C_VEL
LIN {X 0,Y 114.244,Z 605.468,A -85,B 0,C 180,E1 -26953.794,E2 -26953.794} C_VEL
LIN {X 0,Y 121.938,Z 596.949,A -85,B 0,C 180,E1 -26958.527,E2 -26958.527} C_VEL
LIN {X 0,Y 129.164,Z 588.029,A -85,B 0,C 180,E1 -26962.089,E2 -26962.089} C_VEL
LIN {X 0,Y 136.827,Z 577.221,A -85,B 0,C 180,E1 -26965.268,E2 -26965.268} C_VEL
LIN {X 0,Y 138.091,Z 574.89,A -85,B 0,C 180,E1 -26965.955,E2 -26965.955} C_VEL
LIN {X 0,Y 137.62,Z 573.899,A -85,B 0,C 180,E1 -26966.879,E2 -26966.879} C_VEL
LIN {X 0,Y 128.25,Z 577.328,A -85,B 0,C 180,E1 -26971.257,E2 -26971.257} C_VEL
LIN {X 0,Y 116.915,Z 581.19,A -85,B 0,C 180,E1 -26978.858,E2 -26978.858} C_VEL
LIN {X 0,Y 102.752,Z 587.808,A -85,B 0,C 180,E1 -27000,E2 -27000} C_VEL
LIN {X 0,Y 102.112,Z 589.386,A -85,B 0,C 180,E1 -27007.912,E2 -27007.912} C_VEL
LIN {X 0,Y 103.174,Z 591.201,A -85,B 0,C 180,E1 -27015.811,E2 -27015.811} C_VEL
LIN {X 0,Y 106.728,Z 592.391,A -85,B 0,C 180,E1 -27023.272,E2 -27023.272} C_VEL
LIN {X 0,Y 111.445,Z 594.02,A -85,B 0,C 180,E1 -27030.298,E2 -27030.298} C_VEL
LIN {X 0,Y 118.303,Z 595.008,A -85,B 0,C 180,E1 -27036.446,E2 -27036.446} C_VEL
LIN {X 0,Y 123.479,Z 595.339,A -85,B 0,C 180,E1 -27039.815,E2 -27039.815} C_VEL
LIN {X 0,Y 122.617,Z 596.892,A -85,B 0,C 180,E1 -27040.689,E2 -27040.689} C_VEL
LIN {X 0,Y 115.966,Z 604.48,A -85,B 0,C 180,E1 -27044.594,E2 -27044.594} C_VEL
LIN {X 0,Y 108.815,Z 611.829,A -85,B 0,C 180,E1 -27049.769,E2 -27049.769} C_VEL
LIN {X 0,Y 103.628,Z 616.879,A -85,B 0,C 180,E1 -27054.7,E2 -27054.7} C_VEL
LIN {X 0,Y 99.116,Z 621.069,A -85,B 0,C 180,E1 -27060.241,E2 -27060.241} C_VEL
LIN {X 0,Y 94.514,Z 625.228,A -85,B 0,C 180,E1 -27068.173,E2 -27068.173} C_VEL
LIN {X 0,Y 91.853,Z 627.946,A -85,B 0,C 180,E1 -27076.73,E2 -27076.73} C_VEL
LIN {X 0,Y 90.876,Z 629.293,A -85,B 0,C 180,E1 -27085.565,E2 -27085.565} C_VEL
LIN {X 0,Y 90.912,Z 629.457,A -85,B 0,C 180,E1 -27090,E2 -27090} C_VEL
LIN {X 0,Y 90.876,Z 629.28,A -85,B 0,C 180,E1 -27094.435,E2 -27094.435} C_VEL
LIN {X 0,Y 91.851,Z 627.912,A -85,B 0,C 180,E1 -27103.27,E2 -27103.27} C_VEL
LIN {X 0,Y 94.503,Z 625.173,A -85,B 0,C 180,E1 -27111.829,E2 -27111.829} C_VEL
LIN {X 0,Y 99.076,Z 620.986,A -85,B 0,C 180,E1 -27119.772,E2 -27119.772} C_VEL
LIN {X 0,Y 105.145,Z 615.227,A -85,B 0,C 180,E1 -27126.983,E2 -27126.983} C_VEL
LIN {X 0,Y 111.725,Z 608.724,A -85,B 0,C 180,E1 -27132.549,E2 -27132.549} C_VEL
LIN {X 0,Y 119.196,Z 600.63,A -85,B 0,C 180,E1 -27137.478,E2 -27137.478} C_VEL
LIN {X 0,Y 126.32,Z 592.144,A -85,B 0,C 180,E1 -27141.161,E2 -27141.161} C_VEL
LIN {X 0,Y 133.803,Z 581.843,A -85,B 0,C 180,E1 -27144.502,E2 -27144.502} C_VEL
LIN {X 0,Y 138.447,Z 572.622,A -85,B 0,C 180,E1 -27147.558,E2 -27147.558} C_VEL
LIN {X 0,Y 141.158,Z 565.869,A -85,B 0,C 180,E1 -27149.657,E2 -27149.657} C_VEL
LIN {X 0,Y 143.063,Z 558.734,A -85,B 0,C 180,E1 -27152.16,E2 -27152.16} C_VEL
LIN {X 0,Y 144.774,Z 549.308,A -85,B 0,C 180,E1 -27155.632,E2 -27155.632} C_VEL
LIN {X 0,Y 145.074,Z 545.602,A -85,B 0,C 180,E1 -27157.198,E2 -27157.198} C_VEL
LIN {X 0,Y 144.533,Z 540.899,A -85,B 0,C 180,E1 -27160.1,E2 -27160.1} C_VEL
LIN {X 0,Y 144.207,Z 538.929,A -85,B 0,C 180,E1 -27161.532,E2 -27161.532} C_VEL
LIN {X 0,Y 142.981,Z 536.044,A -85,B 0,C 180,E1 -27164.757,E2 -27164.757} C_VEL
LIN {X 0,Y 141.15,Z 531.887,A -85,B 0,C 180,E1 -27171.41,E2 -27171.41} C_VEL
LIN {X 0,Y 140.189,Z 530.572,A -85,B 0,C 180,E1 -27177.127,E2 -27177.127} C_VEL
LIN {X 0,Y 140.04,Z 530.464,A -85,B 0,C 180,E1 -27180,E2 -27180} C_VEL
LIN {X 0,Y 140.128,Z 532.088,A -85,B 0,C 180,E1 -27185.757,E2 -27185.757} C_VEL
LIN {X 0,Y 140.329,Z 534.228,A -85,B 0,C 180,E1 -27189.122,E2 -27189.122} C_VEL
LIN {X 0,Y 140.439,Z 536.41,A -85,B 0,C 180,E1 -27191.362,E2 -27191.362} C_VEL
LIN {X 0,Y 140.159,Z 539.541,A -85,B 0,C 180,E1 -27193.426,E2 -27193.426} C_VEL
LIN {X 0,Y 138.938,Z 549.232,A -85,B 0,C 180,E1 -27198.714,E2 -27198.714} C_VEL
LIN {X 0,Y 138.921,Z 551.315,A -85,B 0,C 180,E1 -27200.145,E2 -27200.145} C_VEL
LIN {X 0,Y 139.102,Z 556.748,A -85,B 0,C 180,E1 -27203.841,E2 -27203.841} C_VEL
LIN {X 0,Y 139.059,Z 559.373,A -85,B 0,C 180,E1 -27205.44,E2 -27205.44} C_VEL
LIN {X 0,Y 138.814,Z 561.132,A -85,B 0,C 180,E1 -27206.295,E2 -27206.295} C_VEL
LIN {X 0,Y 135.652,Z 570.443,A -85,B 0,C 180,E1 -27209.797,E2 -27209.797} C_VEL
LIN {X 0,Y 132.951,Z 576.855,A -85,B 0,C 180,E1 -27212.244,E2 -27212.244} C_VEL
LIN {X 0,Y 126.297,Z 586.092,A -85,B 0,C 180,E1 -27214.836,E2 -27214.836} C_VEL
LIN {X 0,Y 118.652,Z 595.37,A -85,B 0,C 180,E1 -27218.296,E2 -27218.296} C_VEL
LIN {X 0,Y 110.396,Z 604.186,A -85,B 0,C 180,E1 -27222.937,E2 -27222.937} C_VEL
LIN {X 0,Y 103.892,Z 610.403,A -85,B 0,C 180,E1 -27227.431,E2 -27227.431} C_VEL
LIN {X 0,Y 98.23,Z 615.496,A -85,B 0,C 180,E1 -27232.544,E2 -27232.544} C_VEL
LIN {X 0,Y 93.431,Z 619.619,A -85,B 0,C 180,E1 -27238.227,E2 -27238.227} C_VEL
LIN {X 0,Y 88.283,Z 623.774,A -85,B 0,C 180,E1 -27246.544,E2 -27246.544} C_VEL
LIN {X 0,Y 85.139,Z 626.487,A -85,B 0,C 180,E1 -27255.662,E2 -27255.662} C_VEL
LIN {X 0,Y 83.804,Z 627.84,A -85,B 0,C 180,E1 -27265.189,E2 -27265.189} C_VEL
LIN {X 0,Y 83.813,Z 628.016,A -85,B 0,C 180,E1 -27270,E2 -27270} C_VEL
LIN {X 0,Y 84.232,Z 627.371,A -85,B 0,C 180,E1 -27279.606,E2 -27279.606} C_VEL
LIN {X 0,Y 86.457,Z 625.377,A -85,B 0,C 180,E1 -27288.975,E2 -27288.975} C_VEL
LIN {X 0,Y 90.546,Z 621.994,A -85,B 0,C 180,E1 -27297.756,E2 -27297.756} C_VEL
LIN {X 0,Y 94.915,Z 618.517,A -85,B 0,C 180,E1 -27303.734,E2 -27303.734} C_VEL
LIN {X 0,Y 100.617,Z 613.551,A -85,B 0,C 180,E1 -27309.794,E2 -27309.794} C_VEL
LIN {X 0,Y 108.102,Z 606.626,A -85,B 0,C 180,E1 -27315.655,E2 -27315.655} C_VEL
LIN {X 0,Y 116.147,Z 598.34,A -85,B 0,C 180,E1 -27320.488,E2 -27320.488} C_VEL
LIN {X 0,Y 123.624,Z 589.687,A -85,B 0,C 180,E1 -27324.107,E2 -27324.107} C_VEL
LIN {X 0,Y 129.453,Z 582.165,A -85,B 0,C 180,E1 -27326.502,E2 -27326.502} C_VEL
LIN {X 0,Y 129.876,Z 580.816,A -85,B 0,C 180,E1 -27327.239,E2 -27327.239} C_VEL
LIN {X 0,Y 116.051,Z 585.168,A -85,B 0,C 180,E1 -27334.918,E2 -27334.918} C_VEL
LIN {X 0,Y 97.434,Z 592.602,A -85,B 0,C 180,E1 -27360,E2 -27360} C_VEL
LIN {X 0,Y 97.964,Z 595.813,A -85,B 0,C 180,E1 -27376.676,E2 -27376.676} C_VEL
LIN {X 0,Y 101.645,Z 596.991,A -85,B 0,C 180,E1 -27384.51,E2 -27384.51} C_VEL
LIN {X 0,Y 106.674,Z 598.494,A -85,B 0,C 180,E1 -27391.807,E2 -27391.807} C_VEL
LIN {X 0,Y 114.927,Z 599.456,A -85,B 0,C 180,E1 -27398.815,E2 -27398.815} C_VEL
LIN {X 0,Y 114.529,Z 600.763,A -85,B 0,C 180,E1 -27399.92,E2 -27399.92} C_VEL
LIN {X 0,Y 106.627,Z 608.804,A -85,B 0,C 180,E1 -27404.883,E2 -27404.883} C_VEL
LIN {X 0,Y 99.597,Z 615.281,A -85,B 0,C 180,E1 -27410.574,E2 -27410.574} C_VEL
LIN {X 0,Y 94.523,Z 619.767,A -85,B 0,C 180,E1 -27416.107,E2 -27416.107} C_VEL
LIN {X 0,Y 90.253,Z 623.279,A -85,B 0,C 180,E1 -27422.146,E2 -27422.146} C_VEL
LIN {X 0,Y 86.198,Z 626.703,A -85,B 0,C 180,E1 -27430.966,E2 -27430.966} C_VEL
LIN {X 0,Y 84.145,Z 628.731,A -85,B 0,C 180,E1 -27440.384,E2 -27440.384} C_VEL
LIN {X 0,Y 83.792,Z 629.234,A -85,B 0,C 180,E1 -27445.189,E2 -27445.189} C_VEL
LIN {X 0,Y 83.811,Z 629.399,A -85,B 0,C 180,E1 -27450,E2 -27450} C_VEL
LIN {X 0,Y 83.792,Z 629.221,A -85,B 0,C 180,E1 -27454.811,E2 -27454.811} C_VEL
LIN {X 0,Y 84.937,Z 627.853,A -85,B 0,C 180,E1 -27464.373,E2 -27464.373} C_VEL
LIN {X 0,Y 87.911,Z 625.114,A -85,B 0,C 180,E1 -27473.561,E2 -27473.561} C_VEL
LIN {X 0,Y 92.932,Z 620.927,A -85,B 0,C 180,E1 -27481.964,E2 -27481.964} C_VEL
LIN {X 0,Y 99.525,Z 615.168,A -85,B 0,C 180,E1 -27489.46,E2 -27489.46} C_VEL
LIN {X 0,Y 106.59,Z 608.666,A -85,B 0,C 180,E1 -27495.137,E2 -27495.137} C_VEL
LIN {X 0,Y 114.486,Z 600.573,A -85,B 0,C 180,E1 -27500.116,E2 -27500.116} C_VEL
LIN {X 0,Y 121.989,Z 592.089,A -85,B 0,C 180,E1 -27503.762,E2 -27503.762} C_VEL
LIN {X 0,Y 129.139,Z 582.755,A -85,B 0,C 180,E1 -27506.797,E2 -27506.797} C_VEL
LIN {X 0,Y 134.05,Z 573.653,A -85,B 0,C 180,E1 -27509.891,E2 -27509.891} C_VEL
LIN {X 0,Y 136.167,Z 569.075,A -85,B 0,C 180,E1 -27511.333,E2 -27511.333} C_VEL
LIN {X 0,Y 138.625,Z 561.628,A -85,B 0,C 180,E1 -27514.072,E2 -27514.072} C_VEL
LIN {X 0,Y 140.505,Z 553.557,A -85,B 0,C 180,E1 -27517.199,E2 -27517.199} C_VEL
LIN {X 0,Y 141.057,Z 550.579,A -85,B 0,C 180,E1 -27518.445,E2 -27518.445} C_VEL
LIN {X 0,Y 140.815,Z 545.937,A -85,B 0,C 180,E1 -27521.492,E2 -27521.492} C_VEL
LIN {X 0,Y 140.674,Z 544.589,A -85,B 0,C 180,E1 -27522.557,E2 -27522.557} C_VEL
LIN {X 0,Y 139.79,Z 542.159,A -85,B 0,C 180,E1 -27525.441,E2 -27525.441} C_VEL
LIN {X 0,Y 138.449,Z 538.675,A -85,B 0,C 180,E1 -27531.241,E2 -27531.241} C_VEL
LIN {X 0,Y 137.96,Z 537.704,A -85,B 0,C 180,E1 -27534.153,E2 -27534.153} C_VEL
LIN {X 0,Y 137.609,Z 537.204,A -85,B 0,C 180,E1 -27537.073,E2 -27537.073} C_VEL
LIN {X 0,Y 137.453,Z 537.11,A -85,B 0,C 180,E1 -27540,E2 -27540} C_VEL
LIN {X 0,Y 137.353,Z 537.759,A -85,B 0,C 180,E1 -27542.933,E2 -27542.933} C_VEL
LIN {X 0,Y 137.367,Z 538.901,A -85,B 0,C 180,E1 -27545.873,E2 -27545.873} C_VEL
LIN {X 0,Y 137.807,Z 542.678,A -85,B 0,C 180,E1 -27551.771,E2 -27551.771} C_VEL
LIN {X 0,Y 138.406,Z 546.494,A -85,B 0,C 180,E1 -27556.066,E2 -27556.066} C_VEL
LIN {X 0,Y 138.921,Z 551.315,A -85,B 0,C 180,E1 -27560.145,E2 -27560.145} C_VEL
LIN {X 0,Y 138.706,Z 553.647,A -85,B 0,C 180,E1 -27561.439,E2 -27561.439} C_VEL
LIN {X 0,Y 137.831,Z 556.58,A -85,B 0,C 180,E1 -27562.485,E2 -27562.485} C_VEL
LIN {X 0,Y 134.073,Z 565.259,A -85,B 0,C 180,E1 -27564.854,E2 -27564.854} C_VEL
LIN {X 0,Y 133.201,Z 567.295,A -85,B 0,C 180,E1 -27565.567,E2 -27565.567} C_VEL
LIN {X 0,Y 129.996,Z 574.822,A -85,B 0,C 180,E1 -27568.538,E2 -27568.538} C_VEL
LIN {X 0,Y 128.035,Z 578.706,A -85,B 0,C 180,E1 -27570.057,E2 -27570.057} C_VEL
LIN {X 0,Y 119.658,Z 589.405,A -85,B 0,C 180,E1 -27573.18,E2 -27573.18} C_VEL
LIN {X 0,Y 111.84,Z 598.114,A -85,B 0,C 180,E1 -27576.754,E2 -27576.754} C_VEL
LIN {X 0,Y 103.281,Z 606.452,A -85,B 0,C 180,E1 -27581.537,E2 -27581.537} C_VEL
LIN {X 0,Y 96.615,Z 612.251,A -85,B 0,C 180,E1 -27586.286,E2 -27586.286} C_VEL
LIN {X 0,Y 89.104,Z 618.432,A -85,B 0,C 180,E1 -27593.732,E2 -27593.732} C_VEL
LIN {X 0,Y 84.371,Z 621.943,A -85,B 0,C 180,E1 -27600.014,E2 -27600.014} C_VEL
LIN {X 0,Y 79.762,Z 625.364,A -85,B 0,C 180,E1 -27609.363,E2 -27609.363} C_VEL
LIN {X 0,Y 77.238,Z 627.389,A -85,B 0,C 180,E1 -27619.515,E2 -27619.515} C_VEL
LIN {X 0,Y 76.734,Z 628.074,A -85,B 0,C 180,E1 -27630,E2 -27630} C_VEL
LIN {X 0,Y 77.238,Z 627.429,A -85,B 0,C 180,E1 -27640.485,E2 -27640.485} C_VEL
LIN {X 0,Y 79.74,Z 625.435,A -85,B 0,C 180,E1 -27650.643,E2 -27650.643} C_VEL
LIN {X 0,Y 84.32,Z 622.051,A -85,B 0,C 180,E1 -27660.006,E2 -27660.006} C_VEL
LIN {X 0,Y 89.053,Z 618.573,A -85,B 0,C 180,E1 -27666.292,E2 -27666.292} C_VEL
LIN {X 0,Y 94.791,Z 613.966,A -85,B 0,C 180,E1 -27672.146,E2 -27672.146} C_VEL
LIN {X 0,Y 102.098,Z 607.702,A -85,B 0,C 180,E1 -27677.73,E2 -27677.73} C_VEL
LIN {X 0,Y 110.493,Z 599.712,A -85,B 0,C 180,E1 -27682.662,E2 -27682.662} C_VEL
LIN {X 0,Y 118.249,Z 591.328,A -85,B 0,C 180,E1 -27686.313,E2 -27686.313} C_VEL
LIN {X 0,Y 120.664,Z 588.462,A -85,B 0,C 180,E1 -27687.302,E2 -27687.302} C_VEL
LIN {X 0,Y 121.145,Z 587.386,A -85,B 0,C 180,E1 -27687.988,E2 -27687.988} C_VEL
LIN {X 0,Y 107.292,Z 591.262,A -85,B 0,C 180,E1 -27696.857,E2 -27696.857} C_VEL
LIN {X 0,Y 91.873,Z 597.151,A -85,B 0,C 180,E1 -27720,E2 -27720} C_VEL
LIN {X 0,Y 92.568,Z 600.164,A -85,B 0,C 180,E1 -27737.679,E2 -27737.679} C_VEL
LIN {X 0,Y 96.423,Z 601.315,A -85,B 0,C 180,E1 -27745.933,E2 -27745.933} C_VEL
LIN {X 0,Y 101.806,Z 602.701,A -85,B 0,C 180,E1 -27753.522,E2 -27753.522} C_VEL
LIN {X 0,Y 106.496,Z 603.297,A -85,B 0,C 180,E1 -27757.831,E2 -27757.831} C_VEL
LIN {X 0,Y 106.405,Z 604.392,A -85,B 0,C 180,E1 -27759.121,E2 -27759.121} C_VEL
LIN {X 0,Y 98.358,Z 611.718,A -85,B 0,C 180,E1 -27764.395,E2 -27764.395} C_VEL
LIN {X 0,Y 92.273,Z 616.807,A -85,B 0,C 180,E1 -27769.61,E2 -27769.61} C_VEL
LIN {X 0,Y 86.995,Z 620.955,A -85,B 0,C 180,E1 -27775.562,E2 -27775.562} C_VEL
LIN {X 0,Y 81.425,Z 625.112,A -85,B 0,C 180,E1 -27784.433,E2 -27784.433} C_VEL
LIN {X 0,Y 78.043,Z 627.829,A -85,B 0,C 180,E1 -27794.326,E2 -27794.326} C_VEL
LIN {X 0,Y 76.712,Z 629.176,A -85,B 0,C 180,E1 -27804.743,E2 -27804.743} C_VEL
LIN {X 0,Y 76.733,Z 629.34,A -85,B 0,C 180,E1 -27810,E2 -27810} C_VEL
LIN {X 0,Y 77.128,Z 628.646,A -85,B 0,C 180,E1 -27820.5,E2 -27820.5} C_VEL
LIN {X 0,Y 79.473,Z 626.599,A -85,B 0,C 180,E1 -27830.716,E2 -27830.716} C_VEL
LIN {X 0,Y 83.994,Z 623.15,A -85,B 0,C 180,E1 -27840.135,E2 -27840.135} C_VEL
LIN {X 0,Y 90.347,Z 618.195,A -85,B 0,C 180,E1 -27848.485,E2 -27848.485} C_VEL
LIN {X 0,Y 96.17,Z 613.391,A -85,B 0,C 180,E1 -27853.968,E2 -27853.968} C_VEL
LIN {X 0,Y 104.002,Z 606.448,A -85,B 0,C 180,E1 -27859.484,E2 -27859.484} C_VEL
LIN {X 0,Y 112.614,Z 597.829,A -85,B 0,C 180,E1 -27864.224,E2 -27864.224} C_VEL
LIN {X 0,Y 120.635,Z 588.804,A -85,B 0,C 180,E1 -27867.645,E2 -27867.645} C_VEL
LIN {X 0,Y 124.72,Z 583.577,A -85,B 0,C 180,E1 -27869.268,E2 -27869.268} C_VEL
LIN {X 0,Y 130.469,Z 573.599,A -85,B 0,C 180,E1 -27872.724,E2 -27872.724} C_VEL
LIN {X 0,Y 132.569,Z 569.019,A -85,B 0,C 180,E1 -27874.322,E2 -27874.322} C_VEL
LIN {X 0,Y 135.325,Z 561.033,A -85,B 0,C 180,E1 -27877.481,E2 -27877.481} C_VEL
LIN {X 0,Y 136.923,Z 555.113,A -85,B 0,C 180,E1 -27879.948,E2 -27879.948} C_VEL
LIN {X 0,Y 137.03,Z 551.961,A -85,B 0,C 180,E1 -27882.078,E2 -27882.078} C_VEL
LIN {X 0,Y 136.958,Z 550.13,A -85,B 0,C 180,E1 -27883.607,E2 -27883.607} C_VEL
LIN {X 0,Y 136.613,Z 548.882,A -85,B 0,C 180,E1 -27885.095,E2 -27885.095} C_VEL
LIN {X 0,Y 135.424,Z 545.32,A -85,B 0,C 180,E1 -27891.044,E2 -27891.044} C_VEL
LIN {X 0,Y 135.033,Z 544.234,A -85,B 0,C 180,E1 -27894.025,E2 -27894.025} C_VEL
LIN {X 0,Y 134.725,Z 543.687,A -85,B 0,C 180,E1 -27897.01,E2 -27897.01} C_VEL
LIN {X 0,Y 134.56,Z 543.606,A -85,B 0,C 180,E1 -27900,E2 -27900} C_VEL
LIN {X 0,Y 134.381,Z 544.316,A -85,B 0,C 180,E1 -27902.998,E2 -27902.998} C_VEL
LIN {X 0,Y 134.27,Z 545.588,A -85,B 0,C 180,E1 -27906.009,E2 -27906.009} C_VEL
LIN {X 0,Y 134.37,Z 548.356,A -85,B 0,C 180,E1 -27910.548,E2 -27910.548} C_VEL
LIN {X 0,Y 134.676,Z 552.124,A -85,B 0,C 180,E1 -27915.125,E2 -27915.125} C_VEL
LIN {X 0,Y 134.833,Z 556.679,A -85,B 0,C 180,E1 -27919.21,E2 -27919.21} C_VEL
LIN {X 0,Y 134.578,Z 562.101,A -85,B 0,C 180,E1 -27923.059,E2 -27923.059} C_VEL
LIN {X 0,Y 134.468,Z 563.367,A -85,B 0,C 180,E1 -27923.895,E2 -27923.895} C_VEL
LIN {X 0,Y 133.489,Z 566.588,A -85,B 0,C 180,E1 -27925.289,E2 -27925.289} C_VEL
LIN {X 0,Y 133.201,Z 567.295,A -85,B 0,C 180,E1 -27925.567,E2 -27925.567} C_VEL
LIN {X 0,Y 131.663,Z 570.322,A -85,B 0,C 180,E1 -27926.457,E2 -27926.457} C_VEL
LIN {X 0,Y 129.534,Z 573.424,A -85,B 0,C 180,E1 -27927.018,E2 -27927.018} C_VEL
LIN {X 0,Y 121.794,Z 582.548,A -85,B 0,C 180,E1 -27928.229,E2 -27928.229} C_VEL
LIN {X 0,Y 120.968,Z 583.511,A -85,B 0,C 180,E1 -27928.46,E2 -27928.46} C_VEL
LIN {X 0,Y 113.098,Z 592.552,A -85,B 0,C 180,E1 -27931.302,E2 -27931.302} C_VEL
LIN {X 0,Y 103.783,Z 601.955,A -85,B 0,C 180,E1 -27935.647,E2 -27935.647} C_VEL
LIN {X 0,Y 96.253,Z 608.551,A -85,B 0,C 180,E1 -27939.944,E2 -27939.944} C_VEL
LIN {X 0,Y 87.807,Z 615.21,A -85,B 0,C 180,E1 -27946.332,E2 -27946.332} C_VEL
LIN {X 0,Y 81.652,Z 619.737,A -85,B 0,C 180,E1 -27952.95,E2 -27952.95} C_VEL
LIN {X 0,Y 75.4,Z 623.893,A -85,B 0,C 180,E1 -27962.222,E2 -27962.222} C_VEL
LIN {X 0,Y 71.432,Z 626.605,A -85,B 0,C 180,E1 -27972.833,E2 -27972.833} C_VEL
LIN {X 0,Y 69.662,Z 627.957,A -85,B 0,C 180,E1 -27984.21,E2 -27984.21} C_VEL
LIN {X 0,Y 69.646,Z 628.133,A -85,B 0,C 180,E1 -27990,E2 -27990} C_VEL
LIN {X 0,Y 70.249,Z 627.487,A -85,B 0,C 180,E1 -28001.542,E2 -28001.542} C_VEL
LIN {X 0,Y 73.111,Z 625.493,A -85,B 0,C 180,E1 -28012.613,E2 -28012.613} C_VEL
LIN {X 0,Y 78.244,Z 622.108,A -85,B 0,C 180,E1 -28022.611,E2 -28022.611} C_VEL
LIN {X 0,Y 85.332,Z 617.229,A -85,B 0,C 180,E1 -28031.215,E2 -28031.215} C_VEL
LIN {X 0,Y 91.599,Z 612.494,A -85,B 0,C 180,E1 -28036.794,E2 -28036.794} C_VEL
LIN {X 0,Y 99.918,Z 605.63,A -85,B 0,C 180,E1 -28042.307,E2 -28042.307} C_VEL
LIN {X 0,Y 108.95,Z 597.106,A -85,B 0,C 180,E1 -28046.991,E2 -28046.991} C_VEL
LIN {X 0,Y 110.728,Z 595.342,A -85,B 0,C 180,E1 -28047.757,E2 -28047.757} C_VEL
LIN {X 0,Y 111.87,Z 593.496,A -85,B 0,C 180,E1 -28048.981,E2 -28048.981} C_VEL
LIN {X 0,Y 94.988,Z 597.816,A -85,B 0,C 180,E1 -28062.785,E2 -28062.785} C_VEL
LIN {X 0,Y 86.114,Z 601.418,A -85,B 0,C 180,E1 -28080,E2 -28080} C_VEL
LIN {X 0,Y 85.75,Z 603.658,A -85,B 0,C 180,E1 -28094.233,E2 -28094.233} C_VEL
LIN {X 0,Y 91.087,Z 605.357,A -85,B 0,C 180,E1 -28107.577,E2 -28107.577} C_VEL
LIN {X 0,Y 96.898,Z 606.611,A -85,B 0,C 180,E1 -28115.467,E2 -28115.467} C_VEL
LIN {X 0,Y 98.307,Z 607.661,A -85,B 0,C 180,E1 -28118.15,E2 -28118.15} C_VEL
LIN {X 0,Y 91.21,Z 613.464,A -85,B 0,C 180,E1 -28122.945,E2 -28122.945} C_VEL
LIN {X 0,Y 84.94,Z 618.241,A -85,B 0,C 180,E1 -28128.553,E2 -28128.553} C_VEL
LIN {X 0,Y 77.927,Z 623.164,A -85,B 0,C 180,E1 -28137.24,E2 -28137.24} C_VEL
LIN {X 0,Y 72.849,Z 626.587,A -85,B 0,C 180,E1 -28147.301,E2 -28147.301} C_VEL
LIN {X 0,Y 70.147,Z 628.614,A -85,B 0,C 180,E1 -28158.441,E2 -28158.441} C_VEL
LIN {X 0,Y 69.644,Z 629.282,A -85,B 0,C 180,E1 -28170,E2 -28170} C_VEL
LIN {X 0,Y 70.146,Z 628.588,A -85,B 0,C 180,E1 -28181.559,E2 -28181.559} C_VEL
LIN {X 0,Y 72.823,Z 626.54,A -85,B 0,C 180,E1 -28192.708,E2 -28192.708} C_VEL
LIN {X 0,Y 77.908,Z 623.091,A -85,B 0,C 180,E1 -28202.769,E2 -28202.769} C_VEL
LIN {X 0,Y 84.852,Z 618.136,A -85,B 0,C 180,E1 -28211.5,E2 -28211.5} C_VEL
LIN {X 0,Y 93.46,Z 611.532,A -85,B 0,C 180,E1 -28218.762,E2 -28218.762} C_VEL
LIN {X 0,Y 102.033,Z 604.145,A -85,B 0,C 180,E1 -28224.032,E2 -28224.032} C_VEL
LIN {X 0,Y 109.995,Z 596.416,A -85,B 0,C 180,E1 -28227.844,E2 -28227.844} C_VEL
LIN {X 0,Y 118.366,Z 587.087,A -85,B 0,C 180,E1 -28231.138,E2 -28231.138} C_VEL
LIN {X 0,Y 121.495,Z 583.016,A -85,B 0,C 180,E1 -28232.434,E2 -28232.434} C_VEL
LIN {X 0,Y 126.951,Z 574,A -85,B 0,C 180,E1 -28235.57,E2 -28235.57} C_VEL
LIN {X 0,Y 130.061,Z 567.135,A -85,B 0,C 180,E1 -28238.291,E2 -28238.291} C_VEL
LIN {X 0,Y 132.658,Z 559.734,A -85,B 0,C 180,E1 -28241.466,E2 -28241.466} C_VEL
LIN {X 0,Y 133.022,Z 557.301,A -85,B 0,C 180,E1 -28243.106,E2 -28243.106} C_VEL
LIN {X 0,Y 133.051,Z 555.562,A -85,B 0,C 180,E1 -28244.686,E2 -28244.686} C_VEL
LIN {X 0,Y 132.076,Z 551.824,A -85,B 0,C 180,E1 -28250.814,E2 -28250.814} C_VEL
LIN {X 0,Y 131.772,Z 550.647,A -85,B 0,C 180,E1 -28253.877,E2 -28253.877} C_VEL
LIN {X 0,Y 131.532,Z 550.022,A -85,B 0,C 180,E1 -28256.937,E2 -28256.937} C_VEL
LIN {X 0,Y 131.351,Z 549.965,A -85,B 0,C 180,E1 -28260,E2 -28260} C_VEL
LIN {X 0,Y 131.072,Z 550.758,A -85,B 0,C 180,E1 -28263.074,E2 -28263.074} C_VEL
LIN {X 0,Y 130.758,Z 553.027,A -85,B 0,C 180,E1 -28267.746,E2 -28267.746} C_VEL
LIN {X 0,Y 130.77,Z 554.983,A -85,B 0,C 180,E1 -28270.842,E2 -28270.842} C_VEL
LIN {X 0,Y 130.722,Z 559.003,A -85,B 0,C 180,E1 -28275.594,E2 -28275.594} C_VEL
LIN {X 0,Y 130.494,Z 562.656,A -85,B 0,C 180,E1 -28278.853,E2 -28278.853} C_VEL
LIN {X 0,Y 129.87,Z 567.315,A -85,B 0,C 180,E1 -28282.26,E2 -28282.26} C_VEL
LIN {X 0,Y 127.433,Z 572.982,A -85,B 0,C 180,E1 -28284.686,E2 -28284.686} C_VEL
LIN {X 0,Y 123.801,Z 579.85,A -85,B 0,C 180,E1 -28287.491,E2 -28287.491} C_VEL
LIN {X 0,Y 120.968,Z 583.511,A -85,B 0,C 180,E1 -28288.46,E2 -28288.46} C_VEL
LIN {X 0,Y 118.276,Z 586.364,A -85,B 0,C 180,E1 -28288.94,E2 -28288.94} C_VEL
LIN {X 0,Y 107.752,Z 594.801,A -85,B 0,C 180,E1 -28289.24,E2 -28289.24} C_VEL
LIN {X 0,Y 104.957,Z 597.232,A -85,B 0,C 180,E1 -28289.98,E2 -28289.98} C_VEL
LIN {X 0,Y 95.78,Z 605.463,A -85,B 0,C 180,E1 -28294.362,E2 -28294.362} C_VEL
LIN {X 0,Y 86.865,Z 612.368,A -85,B 0,C 180,E1 -28299.77,E2 -28299.77} C_VEL
LIN {X 0,Y 80.09,Z 617.142,A -85,B 0,C 180,E1 -28305.411,E2 -28305.411} C_VEL
LIN {X 0,Y 72.406,Z 622.061,A -85,B 0,C 180,E1 -28314.382,E2 -28314.382} C_VEL
LIN {X 0,Y 66.617,Z 625.482,A -85,B 0,C 180,E1 -28325.04,E2 -28325.04} C_VEL
LIN {X 0,Y 63.304,Z 627.507,A -85,B 0,C 180,E1 -28337.171,E2 -28337.171} C_VEL
LIN {X 0,Y 62.547,Z 628.191,A -85,B 0,C 180,E1 -28350,E2 -28350} C_VEL
LIN {X 0,Y 63.302,Z 627.546,A -85,B 0,C 180,E1 -28362.829,E2 -28362.829} C_VEL
LIN {X 0,Y 66.593,Z 625.551,A -85,B 0,C 180,E1 -28374.97,E2 -28374.97} C_VEL
LIN {X 0,Y 72.334,Z 622.165,A -85,B 0,C 180,E1 -28385.659,E2 -28385.659} C_VEL
LIN {X 0,Y 80.11,Z 617.285,A -85,B 0,C 180,E1 -28394.574,E2 -28394.574} C_VEL
LIN {X 0,Y 86.869,Z 612.549,A -85,B 0,C 180,E1 -28400.227,E2 -28400.227} C_VEL
LIN {X 0,Y 95.729,Z 605.684,A -85,B 0,C 180,E1 -28405.683,E2 -28405.683} C_VEL
LIN {X 0,Y 101.698,Z 600.514,A -85,B 0,C 180,E1 -28408.648,E2 -28408.648} C_VEL
LIN {X 0,Y 102.483,Z 599.077,A -85,B 0,C 180,E1 -28410.121,E2 -28410.121} C_VEL
LIN {X 0,Y 81.499,Z 604.697,A -85,B 0,C 180,E1 -28435.053,E2 -28435.053} C_VEL
LIN {X 0,Y 79.92,Z 607.496,A -85,B 0,C 180,E1 -28455.296,E2 -28455.296} C_VEL
LIN {X 0,Y 85.675,Z 609.104,A -85,B 0,C 180,E1 -28469.484,E2 -28469.484} C_VEL
LIN {X 0,Y 89.761,Z 609.928,A -85,B 0,C 180,E1 -28475.292,E2 -28475.292} C_VEL
LIN {X 0,Y 90.204,Z 610.643,A -85,B 0,C 180,E1 -28477,E2 -28477} C_VEL
LIN {X 0,Y 80.831,Z 617.437,A -85,B 0,C 180,E1 -28484.073,E2 -28484.073} C_VEL
LIN {X 0,Y 73.773,Z 622.046,A -85,B 0,C 180,E1 -28491.74,E2 -28491.74} C_VEL
LIN {X 0,Y 68.833,Z 624.997,A -85,B 0,C 180,E1 -28499.302,E2 -28499.302} C_VEL
LIN {X 0,Y 64.438,Z 627.713,A -85,B 0,C 180,E1 -28510.901,E2 -28510.901} C_VEL
LIN {X 0,Y 62.558,Z 629.059,A -85,B 0,C 180,E1 -28523.55,E2 -28523.55} C_VEL
LIN {X 0,Y 62.543,Z 629.223,A -85,B 0,C 180,E1 -28530,E2 -28530} C_VEL
LIN {X 0,Y 63.18,Z 628.528,A -85,B 0,C 180,E1 -28542.855,E2 -28542.855} C_VEL
LIN {X 0,Y 66.282,Z 626.48,A -85,B 0,C 180,E1 -28555.095,E2 -28555.095} C_VEL
LIN {X 0,Y 72.014,Z 623.032,A -85,B 0,C 180,E1 -28565.842,E2 -28565.842} C_VEL
LIN {X 0,Y 79.638,Z 618.077,A -85,B 0,C 180,E1 -28574.91,E2 -28574.91} C_VEL
LIN {X 0,Y 88.917,Z 611.474,A -85,B 0,C 180,E1 -28582.223,E2 -28582.223} C_VEL
LIN {X 0,Y 97.996,Z 604.088,A -85,B 0,C 180,E1 -28587.424,E2 -28587.424} C_VEL
LIN {X 0,Y 106.376,Z 596.36,A -85,B 0,C 180,E1 -28591.092,E2 -28591.092} C_VEL
LIN {X 0,Y 115.089,Z 587.032,A -85,B 0,C 180,E1 -28594.254,E2 -28594.254} C_VEL
LIN {X 0,Y 117.633,Z 583.822,A -85,B 0,C 180,E1 -28595.278,E2 -28595.278} C_VEL
LIN {X 0,Y 122.67,Z 576.191,A -85,B 0,C 180,E1 -28597.986,E2 -28597.986} C_VEL
LIN {X 0,Y 125.754,Z 570.234,A -85,B 0,C 180,E1 -28600.408,E2 -28600.408} C_VEL
LIN {X 0,Y 128.569,Z 563.624,A -85,B 0,C 180,E1 -28603.386,E2 -28603.386} C_VEL
LIN {X 0,Y 128.822,Z 562.547,A -85,B 0,C 180,E1 -28604.17,E2 -28604.17} C_VEL
LIN {X 0,Y 128.951,Z 560.888,A -85,B 0,C 180,E1 -28605.803,E2 -28605.803} C_VEL
LIN {X 0,Y 128.404,Z 558.178,A -85,B 0,C 180,E1 -28610.549,E2 -28610.549} C_VEL
LIN {X 0,Y 128.201,Z 556.903,A -85,B 0,C 180,E1 -28613.706,E2 -28613.706} C_VEL
LIN {X 0,Y 128.017,Z 556.224,A -85,B 0,C 180,E1 -28616.853,E2 -28616.853} C_VEL
LIN {X 0,Y 127.819,Z 556.185,A -85,B 0,C 180,E1 -28620,E2 -28620} C_VEL
LIN {X 0,Y 127.453,Z 557.034,A -85,B 0,C 180,E1 -28623.161,E2 -28623.161} C_VEL
LIN {X 0,Y 126.973,Z 559.252,A -85,B 0,C 180,E1 -28627.694,E2 -28627.694} C_VEL
LIN {X 0,Y 126.785,Z 561.496,A -85,B 0,C 180,E1 -28631.187,E2 -28631.187} C_VEL
LIN {X 0,Y 126.56,Z 563.848,A -85,B 0,C 180,E1 -28634.143,E2 -28634.143} C_VEL
LIN {X 0,Y 126.141,Z 567.025,A -85,B 0,C 180,E1 -28637.239,E2 -28637.239} C_VEL
LIN {X 0,Y 125.267,Z 571.147,A -85,B 0,C 180,E1 -28640.528,E2 -28640.528} C_VEL
LIN {X 0,Y 121.532,Z 578.17,A -85,B 0,C 180,E1 -28643.548,E2 -28643.548} C_VEL
LIN {X 0,Y 119.808,Z 581.018,A -85,B 0,C 180,E1 -28644.746,E2 -28644.746} C_VEL
LIN {X 0,Y 111.034,Z 591.123,A -85,B 0,C 180,E1 -28647.607,E2 -28647.607} C_VEL
LIN {X 0,Y 104.957,Z 597.232,A -85,B 0,C 180,E1 -28649.98,E2 -28649.98} C_VEL
LIN {X 0,Y 100.901,Z 600.769,A -85,B 0,C 180,E1 -28651.37,E2 -28651.37} C_VEL
LIN {X 0,Y 93.041,Z 606.151,A -85,B 0,C 180,E1 -28653.017,E2 -28653.017} C_VEL
LIN {X 0,Y 84.959,Z 611.001,A -85,B 0,C 180,E1 -28655.047,E2 -28655.047} C_VEL
LIN {X 0,Y 80.669,Z 613.635,A -85,B 0,C 180,E1 -28657.167,E2 -28657.167} C_VEL
LIN {X 0,Y 72.911,Z 618.609,A -85,B 0,C 180,E1 -28663.702,E2 -28663.702} C_VEL
LIN {X 0,Y 66.732,Z 622.12,A -85,B 0,C 180,E1 -28670.809,E2 -28670.809} C_VEL
LIN {X 0,Y 60.224,Z 625.541,A -85,B 0,C 180,E1 -28682.174,E2 -28682.174} C_VEL
LIN {X 0,Y 56.382,Z 627.566,A -85,B 0,C 180,E1 -28695.564,E2 -28695.564} C_VEL
LIN {X 0,Y 55.465,Z 628.25,A -85,B 0,C 180,E1 -28710,E2 -28710} C_VEL
LIN {X 0,Y 56.38,Z 627.604,A -85,B 0,C 180,E1 -28724.437,E2 -28724.437} C_VEL
LIN {X 0,Y 60.199,Z 625.609,A -85,B 0,C 180,E1 -28737.839,E2 -28737.839} C_VEL
LIN {X 0,Y 66.671,Z 622.223,A -85,B 0,C 180,E1 -28749.233,E2 -28749.233} C_VEL
LIN {X 0,Y 75.196,Z 617.342,A -85,B 0,C 180,E1 -28758.392,E2 -28758.392} C_VEL
LIN {X 0,Y 82.486,Z 612.605,A -85,B 0,C 180,E1 -28764.04,E2 -28764.04} C_VEL
LIN {X 0,Y 92.861,Z 604.961,A -85,B 0,C 180,E1 -28769.853,E2 -28769.853} C_VEL
LIN {X 0,Y 93.794,Z 603.931,A -85,B 0,C 180,E1 -28770.892,E2 -28770.892} C_VEL
LIN {X 0,Y 75.381,Z 608.458,A -85,B 0,C 180,E1 -28794.65,E2 -28794.65} C_VEL
LIN {X 0,Y 74.998,Z 611.388,A -85,B 0,C 180,E1 -28820.431,E2 -28820.431} C_VEL
LIN {X 0,Y 82.137,Z 612.914,A -85,B 0,C 180,E1 -28834.605,E2 -28834.605} C_VEL
LIN {X 0,Y 81.261,Z 613.984,A -85,B 0,C 180,E1 -28836.245,E2 -28836.245} C_VEL
LIN {X 0,Y 72.566,Z 619.54,A -85,B 0,C 180,E1 -28843.417,E2 -28843.417} C_VEL
LIN {X 0,Y 66.384,Z 623.049,A -85,B 0,C 180,E1 -28850.564,E2 -28850.564} C_VEL
LIN {X 0,Y 59.906,Z 626.471,A -85,B 0,C 180,E1 -28862.013,E2 -28862.013} C_VEL
LIN {X 0,Y 56.267,Z 628.497,A -85,B 0,C 180,E1 -28875.534,E2 -28875.534} C_VEL
LIN {X 0,Y 55.461,Z 629.165,A -85,B 0,C 180,E1 -28890,E2 -28890} C_VEL
LIN {X 0,Y 56.266,Z 628.47,A -85,B 0,C 180,E1 -28904.467,E2 -28904.467} C_VEL
LIN {X 0,Y 59.884,Z 626.421,A -85,B 0,C 180,E1 -28917.998,E2 -28917.998} C_VEL
LIN {X 0,Y 66.347,Z 622.972,A -85,B 0,C 180,E1 -28929.462,E2 -28929.462} C_VEL
LIN {X 0,Y 74.976,Z 617.874,A -85,B 0,C 180,E1 -28938.993,E2 -28938.993} C_VEL
LIN {X 0,Y 84.739,Z 611.415,A -85,B 0,C 180,E1 -28946.035,E2 -28946.035} C_VEL
LIN {X 0,Y 94.341,Z 604.03,A -85,B 0,C 180,E1 -28951.084,E2 -28951.084} C_VEL
LIN {X 0,Y 103.117,Z 596.303,A -85,B 0,C 180,E1 -28954.563,E2 -28954.563} C_VEL
LIN {X 0,Y 112.177,Z 586.977,A -85,B 0,C 180,E1 -28957.534,E2 -28957.534} C_VEL
LIN {X 0,Y 116.347,Z 581.569,A -85,B 0,C 180,E1 -28959.432,E2 -28959.432} C_VEL
LIN {X 0,Y 119.766,Z 576.507,A -85,B 0,C 180,E1 -28961.262,E2 -28961.262} C_VEL
LIN {X 0,Y 123.091,Z 570.366,A -85,B 0,C 180,E1 -28964.01,E2 -28964.01} C_VEL
LIN {X 0,Y 123.864,Z 568.842,A -85,B 0,C 180,E1 -28964.703,E2 -28964.703} C_VEL
LIN {X 0,Y 124.579,Z 567.041,A -85,B 0,C 180,E1 -28965.879,E2 -28965.879} C_VEL
LIN {X 0,Y 124.682,Z 566.076,A -85,B 0,C 180,E1 -28966.97,E2 -28966.97} C_VEL
LIN {X 0,Y 124.437,Z 564.334,A -85,B 0,C 180,E1 -28970.245,E2 -28970.245} C_VEL
LIN {X 0,Y 124.326,Z 562.992,A -85,B 0,C 180,E1 -28973.509,E2 -28973.509} C_VEL
LIN {X 0,Y 124.21,Z 562.245,A -85,B 0,C 180,E1 -28976.757,E2 -28976.757} C_VEL
LIN {X 0,Y 123.985,Z 562.234,A -85,B 0,C 180,E1 -28980,E2 -28980} C_VEL
LIN {X 0,Y 123.518,Z 563.153,A -85,B 0,C 180,E1 -28983.262,E2 -28983.262} C_VEL
LIN {X 0,Y 122.879,Z 565.281,A -85,B 0,C 180,E1 -28987.581,E2 -28987.581} C_VEL
LIN {X 0,Y 122.677,Z 566.627,A -85,B 0,C 180,E1 -28989.897,E2 -28989.897} C_VEL
LIN {X 0,Y 122.184,Z 569.159,A -85,B 0,C 180,E1 -28993.302,E2 -28993.302} C_VEL
LIN {X 0,Y 121.348,Z 572.68,A -85,B 0,C 180,E1 -28996.833,E2 -28996.833} C_VEL
LIN {X 0,Y 120.47,Z 575.113,A -85,B 0,C 180,E1 -28998.711,E2 -28998.711} C_VEL
LIN {X 0,Y 116.096,Z 582.172,A -85,B 0,C 180,E1 -29001.804,E2 -29001.804} C_VEL
LIN {X 0,Y 106.41,Z 592.664,A -85,B 0,C 180,E1 -29004.75,E2 -29004.75} C_VEL
LIN {X 0,Y 97.617,Z 600.851,A -85,B 0,C 180,E1 -29008.122,E2 -29008.122} C_VEL
LIN {X 0,Y 87.792,Z 608.667,A -85,B 0,C 180,E1 -29012.801,E2 -29012.801} C_VEL
LIN {X 0,Y 80.669,Z 613.635,A -85,B 0,C 180,E1 -29017.167,E2 -29017.167} C_VEL
LIN {X 0,Y 76.452,Z 616.128,A -85,B 0,C 180,E1 -29019.604,E2 -29019.604} C_VEL
LIN {X 0,Y 65.29,Z 621.046,A -85,B 0,C 180,E1 -29025.054,E2 -29025.054} C_VEL
LIN {X 0,Y 59.431,Z 623.248,A -85,B 0,C 180,E1 -29029.533,E2 -29029.533} C_VEL
LIN {X 0,Y 57.13,Z 624.159,A -85,B 0,C 180,E1 -29032.56,E2 -29032.56} C_VEL
LIN {X 0,Y 51.397,Z 626.782,A -85,B 0,C 180,E1 -29045.781,E2 -29045.781} C_VEL
LIN {X 0,Y 48.509,Z 628.134,A -85,B 0,C 180,E1 -29061.67,E2 -29061.67} C_VEL
LIN {X 0,Y 48.367,Z 628.308,A -85,B 0,C 180,E1 -29070,E2 -29070} C_VEL
LIN {X 0,Y 49.526,Z 627.662,A -85,B 0,C 180,E1 -29086.488,E2 -29086.488} C_VEL
LIN {X 0,Y 53.998,Z 625.667,A -85,B 0,C 180,E1 -29101.373,E2 -29101.373} C_VEL
LIN {X 0,Y 61.319,Z 622.28,A -85,B 0,C 180,E1 -29113.447,E2 -29113.447} C_VEL
LIN {X 0,Y 70.647,Z 617.398,A -85,B 0,C 180,E1 -29122.735,E2 -29122.735} C_VEL
LIN {X 0,Y 81.296,Z 610.869,A -85,B 0,C 180,E1 -29129.825,E2 -29129.825} C_VEL
LIN {X 0,Y 83.613,Z 609.283,A -85,B 0,C 180,E1 -29131.029,E2 -29131.029} C_VEL
LIN {X 0,Y 84.318,Z 608.454,A -85,B 0,C 180,E1 -29132.257,E2 -29132.257} C_VEL
LIN {X 0,Y 69.098,Z 611.918,A -85,B 0,C 180,E1 -29154.162,E2 -29154.162} C_VEL
LIN {X 0,Y 67.85,Z 614.279,A -85,B 0,C 180,E1 -29178.104,E2 -29178.104} C_VEL
LIN {X 0,Y 73.962,Z 615.516,A -85,B 0,C 180,E1 -29192.894,E2 -29192.894} C_VEL
LIN {X 0,Y 72.839,Z 616.609,A -85,B 0,C 180,E1 -29194.907,E2 -29194.907} C_VEL
LIN {X 0,Y 65.476,Z 620.728,A -85,B 0,C 180,E1 -29201.292,E2 -29201.292} C_VEL
LIN {X 0,Y 57.051,Z 624.882,A -85,B 0,C 180,E1 -29211.98,E2 -29211.98} C_VEL
LIN {X 0,Y 51.142,Z 627.597,A -85,B 0,C 180,E1 -29225.653,E2 -29225.653} C_VEL
LIN {X 0,Y 48.439,Z 628.942,A -85,B 0,C 180,E1 -29241.658,E2 -29241.658} C_VEL
LIN {X 0,Y 48.361,Z 629.106,A -85,B 0,C 180,E1 -29250,E2 -29250} C_VEL
LIN {X 0,Y 49.385,Z 628.41,A -85,B 0,C 180,E1 -29266.536,E2 -29266.536} C_VEL
LIN {X 0,Y 53.679,Z 626.362,A -85,B 0,C 180,E1 -29281.581,E2 -29281.581} C_VEL
LIN {X 0,Y 60.985,Z 622.913,A -85,B 0,C 180,E1 -29293.745,E2 -29293.745} C_VEL
LIN {X 0,Y 70.232,Z 617.959,A -85,B 0,C 180,E1 -29303.183,E2 -29303.183} C_VEL
LIN {X 0,Y 80.959,Z 611.357,A -85,B 0,C 180,E1 -29310.239,E2 -29310.239} C_VEL
LIN {X 0,Y 91.105,Z 603.973,A -85,B 0,C 180,E1 -29315.015,E2 -29315.015} C_VEL
LIN {X 0,Y 100.26,Z 596.247,A -85,B 0,C 180,E1 -29318.247,E2 -29318.247} C_VEL
LIN {X 0,Y 108.761,Z 587.886,A -85,B 0,C 180,E1 -29320.724,E2 -29320.724} C_VEL
LIN {X 0,Y 113.95,Z 581.509,A -85,B 0,C 180,E1 -29322.937,E2 -29322.937} C_VEL
LIN {X 0,Y 116.705,Z 577.615,A -85,B 0,C 180,E1 -29324.477,E2 -29324.477} C_VEL
LIN {X 0,Y 119.15,Z 573.579,A -85,B 0,C 180,E1 -29326.353,E2 -29326.353} C_VEL
LIN {X 0,Y 120.124,Z 571.807,A -85,B 0,C 180,E1 -29327.327,E2 -29327.327} C_VEL
LIN {X 0,Y 120.16,Z 570.318,A -85,B 0,C 180,E1 -29329.894,E2 -29329.894} C_VEL
LIN {X 0,Y 120.163,Z 568.7,A -85,B 0,C 180,E1 -29333.87,E2 -29333.87} C_VEL
LIN {X 0,Y 120.113,Z 568.09,A -85,B 0,C 180,E1 -29336.646,E2 -29336.646} C_VEL
LIN {X 0,Y 119.849,Z 568.117,A -85,B 0,C 180,E1 -29340,E2 -29340} C_VEL
LIN {X 0,Y 119.261,Z 569.116,A -85,B 0,C 180,E1 -29343.379,E2 -29343.379} C_VEL
LIN {X 0,Y 118.384,Z 571.653,A -85,B 0,C 180,E1 -29348.535,E2 -29348.535} C_VEL
LIN {X 0,Y 117.751,Z 573.832,A -85,B 0,C 180,E1 -29351.811,E2 -29351.811} C_VEL
LIN {X 0,Y 116.649,Z 577.152,A -85,B 0,C 180,E1 -29355.424,E2 -29355.424} C_VEL
LIN {X 0,Y 115.936,Z 578.598,A -85,B 0,C 180,E1 -29356.56,E2 -29356.56} C_VEL
LIN {X 0,Y 112.622,Z 583.349,A -85,B 0,C 180,E1 -29358.704,E2 -29358.704} C_VEL
LIN {X 0,Y 103.638,Z 592.72,A -85,B 0,C 180,E1 -29361.184,E2 -29361.184} C_VEL
LIN {X 0,Y 94.475,Z 600.908,A -85,B 0,C 180,E1 -29364.317,E2 -29364.317} C_VEL
LIN {X 0,Y 84.143,Z 608.725,A -85,B 0,C 180,E1 -29368.716,E2 -29368.716} C_VEL
LIN {X 0,Y 75.782,Z 614.195,A -85,B 0,C 180,E1 -29373.42,E2 -29373.42} C_VEL
LIN {X 0,Y 65.801,Z 619.914,A -85,B 0,C 180,E1 -29381.613,E2 -29381.613} C_VEL
LIN {X 0,Y 57.342,Z 624.07,A -85,B 0,C 180,E1 -29392.206,E2 -29392.206} C_VEL
LIN {X 0,Y 57.13,Z 624.159,A -85,B 0,C 180,E1 -29392.56,E2 -29392.56} C_VEL
LIN {X 0,Y 53.797,Z 625.451,A -85,B 0,C 180,E1 -29397.454,E2 -29397.454} C_VEL
LIN {X 0,Y 47.55,Z 627.062,A -85,B 0,C 180,E1 -29406.007,E2 -29406.007} C_VEL
LIN {X 0,Y 43.252,Z 627.884,A -85,B 0,C 180,E1 -29414.44,E2 -29414.44} C_VEL
LIN {X 0,Y 41.431,Z 628.243,A -85,B 0,C 180,E1 -29422.088,E2 -29422.088} C_VEL
LIN {X 0,Y 41.241,Z 628.274,A -85,B 0,C 180,E1 -29424.82,E2 -29424.82} C_VEL
LIN {X 0,Y 41.283,Z 628.367,A -85,B 0,C 180,E1 -29430,E2 -29430} C_VEL
LIN {X 0,Y 42.765,Z 627.72,A -85,B 0,C 180,E1 -29449.189,E2 -29449.189} C_VEL
LIN {X 0,Y 48.04,Z 625.725,A -85,B 0,C 180,E1 -29465.815,E2 -29465.815} C_VEL
LIN {X 0,Y 56.363,Z 622.337,A -85,B 0,C 180,E1 -29478.431,E2 -29478.431} C_VEL
LIN {X 0,Y 66.56,Z 617.455,A -85,B 0,C 180,E1 -29487.641,E2 -29487.641} C_VEL
LIN {X 0,Y 74.139,Z 613.25,A -85,B 0,C 180,E1 -29492.425,E2 -29492.425} C_VEL
LIN {X 0,Y 74.647,Z 612.592,A -85,B 0,C 180,E1 -29493.889,E2 -29493.889} C_VEL
LIN {X 0,Y 62.655,Z 615.076,A -85,B 0,C 180,E1 -29513.559,E2 -29513.559} C_VEL
LIN {X 0,Y 61.675,Z 617.205,A -85,B 0,C 180,E1 -29539.989,E2 -29539.989} C_VEL
LIN {X 0,Y 66.25,Z 618.014,A -85,B 0,C 180,E1 -29551.933,E2 -29551.933} C_VEL
LIN {X 0,Y 56.062,Z 622.934,A -85,B 0,C 180,E1 -29561.222,E2 -29561.222} C_VEL
LIN {X 0,Y 47.758,Z 626.355,A -85,B 0,C 180,E1 -29573.94,E2 -29573.94} C_VEL
LIN {X 0,Y 42.602,Z 628.381,A -85,B 0,C 180,E1 -29590.735,E2 -29590.735} C_VEL
LIN {X 0,Y 41.275,Z 629.048,A -85,B 0,C 180,E1 -29610,E2 -29610} C_VEL
LIN {X 0,Y 42.6,Z 628.351,A -85,B 0,C 180,E1 -29629.266,E2 -29629.266} C_VEL
LIN {X 0,Y 47.74,Z 626.303,A -85,B 0,C 180,E1 -29646.076,E2 -29646.076} C_VEL
LIN {X 0,Y 56.03,Z 622.854,A -85,B 0,C 180,E1 -29658.816,E2 -29658.816} C_VEL
LIN {X 0,Y 66.198,Z 617.9,A -85,B 0,C 180,E1 -29668.14,E2 -29668.14} C_VEL
LIN {X 0,Y 77.663,Z 611.299,A -85,B 0,C 180,E1 -29674.815,E2 -29674.815} C_VEL
LIN {X 0,Y 88.322,Z 603.915,A -85,B 0,C 180,E1 -29679.225,E2 -29679.225} C_VEL
LIN {X 0,Y 97.846,Z 596.191,A -85,B 0,C 180,E1 -29682.121,E2 -29682.121} C_VEL
LIN {X 0,Y 106.785,Z 587.626,A -85,B 0,C 180,E1 -29684.468,E2 -29684.468} C_VEL
LIN {X 0,Y 111.967,Z 581.452,A -85,B 0,C 180,E1 -29686.633,E2 -29686.633} C_VEL
LIN {X 0,Y 114.787,Z 577.554,A -85,B 0,C 180,E1 -29688.414,E2 -29688.414} C_VEL
LIN {X 0,Y 115.612,Z 576.071,A -85,B 0,C 180,E1 -29689.493,E2 -29689.493} C_VEL
LIN {X 0,Y 115.649,Z 574.672,A -85,B 0,C 180,E1 -29693.019,E2 -29693.019} C_VEL
LIN {X 0,Y 115.734,Z 573.745,A -85,B 0,C 180,E1 -29696.519,E2 -29696.519} C_VEL
LIN {X 0,Y 115.436,Z 573.795,A -85,B 0,C 180,E1 -29700,E2 -29700} C_VEL
LIN {X 0,Y 114.684,Z 574.906,A -85,B 0,C 180,E1 -29703.514,E2 -29703.514} C_VEL
LIN {X 0,Y 113.665,Z 577.26,A -85,B 0,C 180,E1 -29708.392,E2 -29708.392} C_VEL
LIN {X 0,Y 113.066,Z 578.738,A -85,B 0,C 180,E1 -29710.747,E2 -29710.747} C_VEL
LIN {X 0,Y 111.986,Z 581.161,A -85,B 0,C 180,E1 -29713.612,E2 -29713.612} C_VEL
LIN {X 0,Y 110.703,Z 583.009,A -85,B 0,C 180,E1 -29714.711,E2 -29714.711} C_VEL
LIN {X 0,Y 109.388,Z 584.66,A -85,B 0,C 180,E1 -29715.479,E2 -29715.479} C_VEL
LIN {X 0,Y 99.672,Z 594.246,A -85,B 0,C 180,E1 -29717.843,E2 -29717.843} C_VEL
LIN {X 0,Y 90.208,Z 602.184,A -85,B 0,C 180,E1 -29720.787,E2 -29720.787} C_VEL
LIN {X 0,Y 80.963,Z 608.783,A -85,B 0,C 180,E1 -29724.293,E2 -29724.293} C_VEL
LIN {X 0,Y 72.096,Z 614.253,A -85,B 0,C 180,E1 -29728.677,E2 -29728.677} C_VEL
LIN {X 0,Y 61.286,Z 619.973,A -85,B 0,C 180,E1 -29736.609,E2 -29736.609} C_VEL
LIN {X 0,Y 51.894,Z 624.129,A -85,B 0,C 180,E1 -29747.378,E2 -29747.378} C_VEL
LIN {X 0,Y 45.008,Z 626.841,A -85,B 0,C 180,E1 -29762.066,E2 -29762.066} C_VEL
LIN {X 0,Y 41.485,Z 628.193,A -85,B 0,C 180,E1 -29780.246,E2 -29780.246} C_VEL
LIN {X 0,Y 41.241,Z 628.274,A -85,B 0,C 180,E1 -29784.82,E2 -29784.82} C_VEL
LIN {X 0,Y 40.883,Z 628.371,A -85,B 0,C 180,E1 -29790.267,E2 -29790.267} C_VEL
LIN {X 0,Y 40.238,Z 628.297,A -85,B 0,C 180,E1 -29795.747,E2 -29795.747} C_VEL
LIN {X 0,Y 38.91,Z 627.946,A -85,B 0,C 180,E1 -29807.103,E2 -29807.103} C_VEL
LIN {X 0,Y 38.86,Z 627.233,A -85,B 0,C 180,E1 -29818.965,E2 -29818.965} C_VEL
LIN {X 0,Y 40.551,Z 626.407,A -85,B 0,C 180,E1 -29827.203,E2 -29827.203} C_VEL
LIN {X 0,Y 41.526,Z 626.055,A -85,B 0,C 180,E1 -29829.604,E2 -29829.604} C_VEL
LIN {X 0,Y 46.865,Z 624.268,A -85,B 0,C 180,E1 -29838.575,E2 -29838.575} C_VEL
LIN {X 0,Y 57.305,Z 620.148,A -85,B 0,C 180,E1 -29849.148,E2 -29849.148} C_VEL
LIN {X 0,Y 65.07,Z 616.524,A -85,B 0,C 180,E1 -29854.403,E2 -29854.403} C_VEL
LIN {X 0,Y 61.951,Z 616.754,A -85,B 0,C 180,E1 -29860.102,E2 -29860.102} C_VEL
LIN {X 0,Y 54.529,Z 618.418,A -85,B 0,C 180,E1 -29879.999,E2 -29879.999} C_VEL
LIN {X 0,Y 55.468,Z 619.812,A -85,B 0,C 180,E1 -29902.34,E2 -29902.34} C_VEL
LIN {X 0,Y 57.76,Z 620.165,A -85,B 0,C 180,E1 -29909.123,E2 -29909.123} C_VEL
LIN {X 0,Y 57.07,Z 620.614,A -85,B 0,C 180,E1 -29910.454,E2 -29910.454} C_VEL
LIN {X 0,Y 46.63,Z 624.766,A -85,B 0,C 180,E1 -29921.098,E2 -29921.098} C_VEL
LIN {X 0,Y 38.594,Z 627.48,A -85,B 0,C 180,E1 -29936.886,E2 -29936.886} C_VEL
LIN {X 0,Y 34.423,Z 628.825,A -85,B 0,C 180,E1 -29958.219,E2 -29958.219} C_VEL
LIN {X 0,Y 34.161,Z 628.989,A -85,B 0,C 180,E1 -29970,E2 -29970} C_VEL
LIN {X 0,Y 35.957,Z 628.292,A -85,B 0,C 180,E1 -29993.011,E2 -29993.011} C_VEL
LIN {X 0,Y 42.175,Z 626.243,A -85,B 0,C 180,E1 -30011.802,E2 -30011.802} C_VEL
LIN {X 0,Y 51.6,Z 622.794,A -85,B 0,C 180,E1 -30024.807,E2 -30024.807} C_VEL
LIN {X 0,Y 62.719,Z 617.841,A -85,B 0,C 180,E1 -30033.695,E2 -30033.695} C_VEL
LIN {X 0,Y 74.909,Z 611.24,A -85,B 0,C 180,E1 -30039.752,E2 -30039.752} C_VEL
LIN {X 0,Y 86.051,Z 603.858,A -85,B 0,C 180,E1 -30043.67,E2 -30043.67} C_VEL
LIN {X 0,Y 95.903,Z 596.134,A -85,B 0,C 180,E1 -30046.166,E2 -30046.166} C_VEL
LIN {X 0,Y 104.252,Z 588.388,A -85,B 0,C 180,E1 -30048.061,E2 -30048.061} C_VEL
LIN {X 0,Y 108.637,Z 583.554,A -85,B 0,C 180,E1 -30049.716,E2 -30049.716} C_VEL
LIN {X 0,Y 110.806,Z 580.785,A -85,B 0,C 180,E1 -30051.127,E2 -30051.127} C_VEL
LIN {X 0,Y 111.063,Z 579.215,A -85,B 0,C 180,E1 -30056.372,E2 -30056.372} C_VEL
LIN {X 0,Y 110.728,Z 579.285,A -85,B 0,C 180,E1 -30060,E2 -30060} C_VEL
LIN {X 0,Y 109.822,Z 580.476,A -85,B 0,C 180,E1 -30063.669,E2 -30063.669} C_VEL
LIN {X 0,Y 108.902,Z 582.181,A -85,B 0,C 180,E1 -30067.416,E2 -30067.416} C_VEL
LIN {X 0,Y 108.285,Z 583.35,A -85,B 0,C 180,E1 -30069.459,E2 -30069.459} C_VEL
LIN {X 0,Y 107.476,Z 584.754,A -85,B 0,C 180,E1 -30071.314,E2 -30071.314} C_VEL
LIN {X 0,Y 106.627,Z 585.834,A -85,B 0,C 180,E1 -30071.982,E2 -30071.982} C_VEL
LIN {X 0,Y 97.732,Z 594.302,A -85,B 0,C 180,E1 -30073.879,E2 -30073.879} C_VEL
LIN {X 0,Y 87.932,Z 602.241,A -85,B 0,C 180,E1 -30076.443,E2 -30076.443} C_VEL
LIN {X 0,Y 78.303,Z 608.841,A -85,B 0,C 180,E1 -30079.538,E2 -30079.538} C_VEL
LIN {X 0,Y 68.959,Z 614.312,A -85,B 0,C 180,E1 -30083.474,E2 -30083.474} C_VEL
LIN {X 0,Y 60.139,Z 618.786,A -85,B 0,C 180,E1 -30088.78,E2 -30088.78} C_VEL
LIN {X 0,Y 51.946,Z 622.297,A -85,B 0,C 180,E1 -30095.732,E2 -30095.732} C_VEL
LIN {X 0,Y 42.481,Z 625.719,A -85,B 0,C 180,E1 -30108.566,E2 -30108.566} C_VEL
LIN {X 0,Y 36.114,Z 627.743,A -85,B 0,C 180,E1 -30127.095,E2 -30127.095} C_VEL
LIN {X 0,Y 34.173,Z 628.426,A -85,B 0,C 180,E1 -30150,E2 -30150} C_VEL
LIN {X 0,Y 36.11,Z 627.779,A -85,B 0,C 180,E1 -30172.908,E2 -30172.908} C_VEL
LIN {X 0,Y 41.526,Z 626.055,A -85,B 0,C 180,E1 -30189.604,E2 -30189.604} C_VEL
LIN {X 0,Y 43.237,Z 625.375,A -85,B 0,C 180,E1 -30194.379,E2 -30194.379} C_VEL
LIN {X 0,Y 45.162,Z 624.133,A -85,B 0,C 180,E1 -30202.611,E2 -30202.611} C_VEL
LIN {X 0,Y 47.863,Z 622.668,A -85,B 0,C 180,E1 -30210.027,E2 -30210.027} C_VEL
LIN {X 0,Y 50.555,Z 621.563,A -85,B 0,C 180,E1 -30213.225,E2 -30213.225} C_VEL
LIN {X 0,Y 53.997,Z 620.205,A -85,B 0,C 180,E1 -30215.656,E2 -30215.656} C_VEL
LIN {X 0,Y 55.65,Z 619.407,A -85,B 0,C 180,E1 -30217.736,E2 -30217.736} C_VEL
LIN {X 0,Y 47.193,Z 621.324,A -85,B 0,C 180,E1 -30248.564,E2 -30248.564} C_VEL
LIN {X 0,Y 49.271,Z 622.096,A -85,B 0,C 180,E1 -30265.335,E2 -30265.335} C_VEL
LIN {X 0,Y 47.862,Z 622.819,A -85,B 0,C 180,E1 -30268.232,E2 -30268.232} C_VEL
LIN {X 0,Y 37.17,Z 626.239,A -85,B 0,C 180,E1 -30280.86,E2 -30280.86} C_VEL
LIN {X 0,Y 29.521,Z 628.264,A -85,B 0,C 180,E1 -30301.567,E2 -30301.567} C_VEL
LIN {X 0,Y 27.054,Z 628.931,A -85,B 0,C 180,E1 -30330,E2 -30330} C_VEL
LIN {X 0,Y 29.518,Z 628.233,A -85,B 0,C 180,E1 -30358.437,E2 -30358.437} C_VEL
LIN {X 0,Y 37.155,Z 626.184,A -85,B 0,C 180,E1 -30379.166,E2 -30379.166} C_VEL
LIN {X 0,Y 47.838,Z 622.735,A -85,B 0,C 180,E1 -30391.822,E2 -30391.822} C_VEL
LIN {X 0,Y 59.9,Z 617.782,A -85,B 0,C 180,E1 -30399.823,E2 -30399.823} C_VEL
LIN {X 0,Y 72.746,Z 611.182,A -85,B 0,C 180,E1 -30405.04,E2 -30405.04} C_VEL
LIN {X 0,Y 84.325,Z 603.8,A -85,B 0,C 180,E1 -30408.322,E2 -30408.322} C_VEL
LIN {X 0,Y 94.457,Z 596.078,A -85,B 0,C 180,E1 -30410.354,E2 -30410.354} C_VEL
LIN {X 0,Y 102.123,Z 589.172,A -85,B 0,C 180,E1 -30411.815,E2 -30411.815} C_VEL
LIN {X 0,Y 104.977,Z 586.272,A -85,B 0,C 180,E1 -30412.755,E2 -30412.755} C_VEL
LIN {X 0,Y 105.956,Z 585.137,A -85,B 0,C 180,E1 -30413.429,E2 -30413.429} C_VEL
LIN {X 0,Y 106.128,Z 584.46,A -85,B 0,C 180,E1 -30416.203,E2 -30416.203} C_VEL
LIN {X 0,Y 105.72,Z 584.583,A -85,B 0,C 180,E1 -30420,E2 -30420} C_VEL
LIN {X 0,Y 104.633,Z 585.857,A -85,B 0,C 180,E1 -30423.852,E2 -30423.852} C_VEL
LIN {X 0,Y 103.454,Z 587.655,A -85,B 0,C 180,E1 -30427.809,E2 -30427.809} C_VEL
LIN {X 0,Y 101.534,Z 589.645,A -85,B 0,C 180,E1 -30428.902,E2 -30428.902} C_VEL
LIN {X 0,Y 91.202,Z 598.512,A -85,B 0,C 180,E1 -30430.731,E2 -30430.731} C_VEL
LIN {X 0,Y 79.524,Z 606.856,A -85,B 0,C 180,E1 -30433.557,E2 -30433.557} C_VEL
LIN {X 0,Y 69.678,Z 612.66,A -85,B 0,C 180,E1 -30436.623,E2 -30436.623} C_VEL
LIN {X 0,Y 60.11,Z 617.437,A -85,B 0,C 180,E1 -30440.715,E2 -30440.715} C_VEL
LIN {X 0,Y 48.136,Z 622.356,A -85,B 0,C 180,E1 -30448.834,E2 -30448.834} C_VEL
LIN {X 0,Y 37.428,Z 625.778,A -85,B 0,C 180,E1 -30461.314,E2 -30461.314} C_VEL
LIN {X 0,Y 29.69,Z 627.802,A -85,B 0,C 180,E1 -30481.743,E2 -30481.743} C_VEL
LIN {X 0,Y 27.068,Z 628.484,A -85,B 0,C 180,E1 -30510,E2 -30510} C_VEL
LIN {X 0,Y 29.684,Z 627.837,A -85,B 0,C 180,E1 -30538.263,E2 -30538.263} C_VEL
LIN {X 0,Y 37.402,Z 625.841,A -85,B 0,C 180,E1 -30558.731,E2 -30558.731} C_VEL
LIN {X 0,Y 48.11,Z 622.451,A -85,B 0,C 180,E1 -30571.221,E2 -30571.221} C_VEL
LIN {X 0,Y 50.555,Z 621.563,A -85,B 0,C 180,E1 -30573.225,E2 -30573.225} C_VEL
LIN {X 0,Y 51.205,Z 621.235,A -85,B 0,C 180,E1 -30574.58,E2 -30574.58} C_VEL
LIN {X 0,Y 50.875,Z 621.034,A -85,B 0,C 180,E1 -30577.439,E2 -30577.439} C_VEL
LIN {X 0,Y 49.133,Z 621.202,A -85,B 0,C 180,E1 -30581.236,E2 -30581.236} C_VEL
LIN {X 0,Y 41.712,Z 622.792,A -85,B 0,C 180,E1 -30595.11,E2 -30595.11} C_VEL
LIN {X 0,Y 41.251,Z 622.911,A -85,B 0,C 180,E1 -30597.383,E2 -30597.383} C_VEL
LIN {X 0,Y 41.135,Z 623.744,A -85,B 0,C 180,E1 -30619.98,E2 -30619.98} C_VEL
LIN {X 0,Y 40.284,Z 624.205,A -85,B 0,C 180,E1 -30623.654,E2 -30623.654} C_VEL
LIN {X 0,Y 32.944,Z 626.181,A -85,B 0,C 180,E1 -30631.425,E2 -30631.425} C_VEL
LIN {X 0,Y 23.498,Z 628.205,A -85,B 0,C 180,E1 -30653.261,E2 -30653.261} C_VEL
LIN {X 0,Y 19.961,Z 628.872,A -85,B 0,C 180,E1 -30690,E2 -30690} C_VEL
LIN {X 0,Y 23.495,Z 628.174,A -85,B 0,C 180,E1 -30726.745,E2 -30726.745} C_VEL
LIN {X 0,Y 32.933,Z 626.125,A -85,B 0,C 180,E1 -30748.607,E2 -30748.607} C_VEL
LIN {X 0,Y 44.908,Z 622.676,A -85,B 0,C 180,E1 -30759.881,E2 -30759.881} C_VEL
LIN {X 0,Y 57.824,Z 617.723,A -85,B 0,C 180,E1 -30766.489,E2 -30766.489} C_VEL
LIN {X 0,Y 71.238,Z 611.124,A -85,B 0,C 180,E1 -30770.594,E2 -30770.594} C_VEL
LIN {X 0,Y 83.176,Z 603.743,A -85,B 0,C 180,E1 -30773.13,E2 -30773.13} C_VEL
LIN {X 0,Y 93.529,Z 596.022,A -85,B 0,C 180,E1 -30774.65,E2 -30774.65} C_VEL
LIN {X 0,Y 100.046,Z 590.339,A -85,B 0,C 180,E1 -30775.607,E2 -30775.607} C_VEL
LIN {X 0,Y 100.954,Z 589.457,A -85,B 0,C 180,E1 -30776.008,E2 -30776.008} C_VEL
LIN {X 0,Y 100.476,Z 589.616,A -85,B 0,C 180,E1 -30780,E2 -30780} C_VEL
LIN {X 0,Y 98.779,Z 591.457,A -85,B 0,C 180,E1 -30785.073,E2 -30785.073} C_VEL
LIN {X 0,Y 88.429,Z 599.906,A -85,B 0,C 180,E1 -30786.56,E2 -30786.56} C_VEL
LIN {X 0,Y 76.46,Z 607.959,A -85,B 0,C 180,E1 -30788.843,E2 -30788.843} C_VEL
LIN {X 0,Y 64.616,Z 614.429,A -85,B 0,C 180,E1 -30791.793,E2 -30791.793} C_VEL
LIN {X 0,Y 54.713,Z 618.904,A -85,B 0,C 180,E1 -30795.552,E2 -30795.552} C_VEL
LIN {X 0,Y 45.134,Z 622.415,A -85,B 0,C 180,E1 -30800.887,E2 -30800.887} C_VEL
LIN {X 0,Y 33.152,Z 625.837,A -85,B 0,C 180,E1 -30812.008,E2 -30812.008} C_VEL
LIN {X 0,Y 23.67,Z 627.861,A -85,B 0,C 180,E1 -30833.57,E2 -30833.57} C_VEL
LIN {X 0,Y 19.976,Z 628.543,A -85,B 0,C 180,E1 -30870,E2 -30870} C_VEL
LIN {X 0,Y 23.664,Z 627.895,A -85,B 0,C 180,E1 -30906.441,E2 -30906.441} C_VEL
LIN {X 0,Y 33.13,Z 625.899,A -85,B 0,C 180,E1 -30928.052,E2 -30928.052} C_VEL
LIN {X 0,Y 45.109,Z 622.509,A -85,B 0,C 180,E1 -30939.197,E2 -30939.197} C_VEL
LIN {X 0,Y 45.509,Z 622.189,A -85,B 0,C 180,E1 -30942.008,E2 -30942.008} C_VEL
LIN {X 0,Y 41.251,Z 622.911,A -85,B 0,C 180,E1 -30957.383,E2 -30957.383} C_VEL
LIN {X 0,Y 40.103,Z 623.271,A -85,B 0,C 180,E1 -30961.821,E2 -30961.821} C_VEL
LIN {X 0,Y 37.45,Z 624.076,A -85,B 0,C 180,E1 -30967.584,E2 -30967.584} C_VEL
LIN {X 0,Y 33.501,Z 625.201,A -85,B 0,C 180,E1 -30973.863,E2 -30973.863} C_VEL
LIN {X 0,Y 28.973,Z 626.309,A -85,B 0,C 180,E1 -30980.155,E2 -30980.155} C_VEL
LIN {X 0,Y 26.557,Z 626.748,A -85,B 0,C 180,E1 -30983.273,E2 -30983.273} C_VEL
LIN {X 0,Y 18.295,Z 628.147,A -85,B 0,C 180,E1 -30999.8,E2 -30999.8} C_VEL
LIN {X 0,Y 12.856,Z 628.813,A -85,B 0,C 180,E1 -31050,E2 -31050} C_VEL
LIN {X 0,Y 18.293,Z 628.115,A -85,B 0,C 180,E1 -31100.211,E2 -31100.211} C_VEL
LIN {X 0,Y 29.845,Z 626.066,A -85,B 0,C 180,E1 -31120.379,E2 -31120.379} C_VEL
LIN {X 0,Y 42.979,Z 622.617,A -85,B 0,C 180,E1 -31128.852,E2 -31128.852} C_VEL
LIN {X 0,Y 56.584,Z 617.664,A -85,B 0,C 180,E1 -31133.536,E2 -31133.536} C_VEL
LIN {X 0,Y 70.425,Z 611.065,A -85,B 0,C 180,E1 -31136.326,E2 -31136.326} C_VEL
LIN {X 0,Y 82.627,Z 603.685,A -85,B 0,C 180,E1 -31138.054,E2 -31138.054} C_VEL
LIN {X 0,Y 92.976,Z 596.093,A -85,B 0,C 180,E1 -31138.995,E2 -31138.995} C_VEL
LIN {X 0,Y 94.892,Z 594.475,A -85,B 0,C 180,E1 -31140,E2 -31140} C_VEL
LIN {X 0,Y 92.991,Z 596.062,A -85,B 0,C 180,E1 -31141.441,E2 -31141.441} C_VEL
LIN {X 0,Y 82.664,Z 603.632,A -85,B 0,C 180,E1 -31142.6,E2 -31142.6} C_VEL
LIN {X 0,Y 70.477,Z 610.986,A -85,B 0,C 180,E1 -31144.28,E2 -31144.28} C_VEL
LIN {X 0,Y 56.654,Z 617.554,A -85,B 0,C 180,E1 -31147.065,E2 -31147.065} C_VEL
LIN {X 0,Y 43.106,Z 622.474,A -85,B 0,C 180,E1 -31151.976,E2 -31151.976} C_VEL
LIN {X 0,Y 29.987,Z 625.896,A -85,B 0,C 180,E1 -31160.368,E2 -31160.368} C_VEL
LIN {X 0,Y 18.425,Z 627.92,A -85,B 0,C 180,E1 -31180.283,E2 -31180.283} C_VEL
LIN {X 0,Y 12.873,Z 628.601,A -85,B 0,C 180,E1 -31230,E2 -31230} C_VEL
LIN {X 0,Y 18.42,Z 627.954,A -85,B 0,C 180,E1 -31279.737,E2 -31279.737} C_VEL
LIN {X 0,Y 29.972,Z 625.957,A -85,B 0,C 180,E1 -31299.706,E2 -31299.706} C_VEL
LIN {X 0,Y 36.44,Z 624.441,A -85,B 0,C 180,E1 -31304.647,E2 -31304.647} C_VEL
LIN {X 0,Y 35.801,Z 624.471,A -85,B 0,C 180,E1 -31308.678,E2 -31308.678} C_VEL
LIN {X 0,Y 33.664,Z 625.189,A -85,B 0,C 180,E1 -31334.459,E2 -31334.459} C_VEL
LIN {X 0,Y 31.998,Z 625.638,A -85,B 0,C 180,E1 -31337.803,E2 -31337.803} C_VEL
LIN {X 0,Y 26.557,Z 626.748,A -85,B 0,C 180,E1 -31343.273,E2 -31343.273} C_VEL
LIN {X 0,Y 21.33,Z 627.634,A -85,B 0,C 180,E1 -31349.575,E2 -31349.575} C_VEL
LIN {X 0,Y 15.918,Z 628.243,A -85,B 0,C 180,E1 -31356.973,E2 -31356.973} C_VEL
LIN {X 0,Y 6.665,Z 628.747,A -85,B 0,C 180,E1 -31400.567,E2 -31400.567} C_VEL
LIN {X 0,Y 8.606,Z 628.58,A -85,B 0,C 180,E1 -31462.285,E2 -31462.285} C_VEL
LIN {X 0,Y 21.412,Z 627.202,A -85,B 0,C 180,E1 -31489.967,E2 -31489.967} C_VEL
LIN {X 0,Y 35.202,Z 624.463,A -85,B 0,C 180,E1 -31496.593,E2 -31496.593} C_VEL
LIN {X 0,Y 49.196,Z 620.277,A -85,B 0,C 180,E1 -31499.794,E2 -31499.794} C_VEL
LIN {X 0,Y 50.342,Z 619.874,A -85,B 0,C 180,E1 -31500.001,E2 -31500.001} C_VEL
LIN {X 0,Y 49.204,Z 620.269,A -85,B 0,C 180,E1 -31501.008,E2 -31501.008} C_VEL
LIN {X 0,Y 35.235,Z 624.424,A -85,B 0,C 180,E1 -31504.213,E2 -31504.213} C_VEL
LIN {X 0,Y 21.483,Z 627.136,A -85,B 0,C 180,E1 -31511.059,E2 -31511.059} C_VEL
LIN {X 0,Y 8.837,Z 628.486,A -85,B 0,C 180,E1 -31537.32,E2 -31537.32} C_VEL
LIN {X 0,Y 5.763,Z 628.66,A -85,B 0,C 180,E1 -31590,E2 -31590} C_VEL
LIN {X 0,Y 14.848,Z 628.012,A -85,B 0,C 180,E1 -31661.204,E2 -31661.204} C_VEL
LIN {X 0,Y 24.293,Z 626.722,A -85,B 0,C 180,E1 -31671.143,E2 -31671.143} C_VEL
LIN {X 0,Y 27.295,Z 626.206,A -85,B 0,C 180,E1 -31676.071,E2 -31676.071} C_VEL
LIN {X 0,Y 26.683,Z 626.347,A -85,B 0,C 180,E1 -31683.655,E2 -31683.655} C_VEL
LIN {X 0,Y 23.839,Z 626.847,A -85,B 0,C 180,E1 -31688.324,E2 -31688.324} C_VEL
LIN {X 0,Y 14.783,Z 628.089,A -85,B 0,C 180,E1 -31698.046,E2 -31698.046} C_VEL
LIN {X 0,Y 5.743,Z 628.755,A -85,B 0,C 180,E1 -31770,E2 -31770} C_VEL
LIN {X 0,Y 8.606,Z 628.58,A -85,B 0,C 180,E1 -31822.285,E2 -31822.285} C_VEL
LIN {X 0,Y 8.606,Z 628.58,A -85,B 0,C 180,E1 -31822.285,E2 -31822.285}

QRS_NEXT_CUT()

QRS_NEXT()
QRS_HOME()

END
